KUKA KRL program: ps_604ac_c1.src, ps_604ac_c1.dat

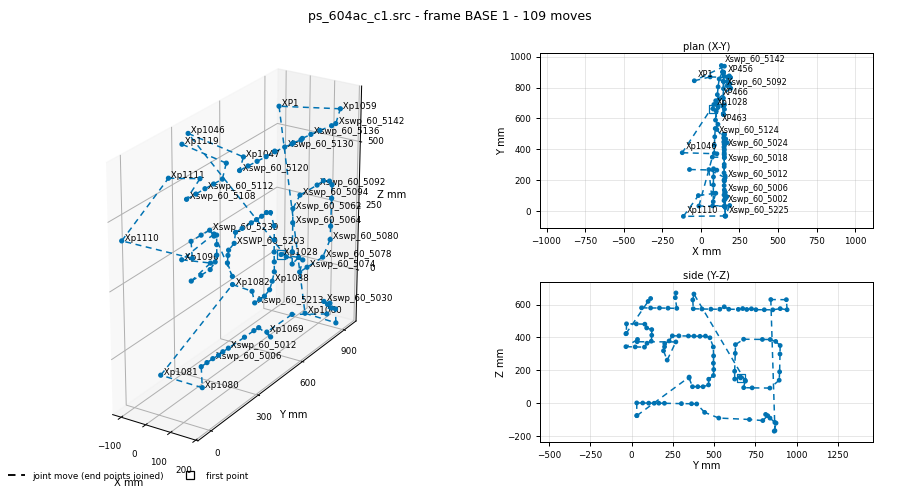
[picture p0: tool path of ps_604ac_c1.src in frame BASE 1, 109 of 111 moves have a stored position in this frame; points joined in program order, loops and branches not executed]
--- ps_604ac_c1.src ---
&ACCESS RVO1
&REL 76
&COMMENT Resp C1 Actros
DEF ps_604ac_c1( )
EXT e_Fraes1 ( )
EXT f_Fraes1 ( )
  ;FOLD INI;%{PE}%V2.2.2,%MKUKATPBASIS,%CINIT,%VCOMMON,%P
  ;FOLD BAS INI;%{PE}%V2.2.2,%MKUKATPBASIS,%CINIT,%VINIT,%P
  INTERRUPT DECL 3 WHEN $STOPMESS==TRUE DO IR_STOPM ( )
  INTERRUPT ON 3
  BAS (#INITMOV,0 )
  ;ENDFOLD
  ;FOLD A20 INI;%{E}%V2.2.2,%MKUKATPA20,%CINIT,%VINIT,%P
  IF ARC20==TRUE THEN
    A20 (ARC_INI)
    INTERRUPT DECL 6 WHEN $CYCFLAG[3]==FALSE DO A20(TECH_STOP2)
  ENDIF
  ;ENDFOLD
  ;FOLD A10 INI;%{E}%V2.2.2,%MKUKATPARC,%CINIT,%VINIT,%P
  IF A10_OPTION==#ACTIVE THEN
    INTERRUPT DECL 4 WHEN $CYCFLAG[2]==FALSE DO A10 (#APPL_ERROR)
    INTERRUPT DECL 7 WHEN A_ARC_SWI==#ACTIVE DO A10 (#ARC_SEAM)
    INTERRUPT DECL 5 WHEN A_FLY_ARC==TRUE DO A10 (#HPU_ARC)
    INTERRUPT  ON 5
    A10_INI ( )
  ENDIF
  ;ENDFOLD
  ;FOLD GRIPPER INI;%{E}%V2.2.2,%MKUKATPGRIPPER,%CINIT,%VINIT,%P
  USER_GRP(0,DUMMY,DUMMY,GDEFAULT)
  ;ENDFOLD
  ;FOLD SPOT INI;%{E}%V.2.2,%MKUKATPSPOT,%CINIT,%VINIT,%P
  USERSPOT(#INIT)
  ;ENDFOLD
  ;FOLD TOUCHSENSE INI;%{E}%V2.2.2,%MKUKATPTS,%CINIT,%VINIT,%P
  IF H70_OPTION THEN
    INTERRUPT DECL 15 WHEN $MEAS_PULSE[TOUCH_I[TOUCH_ACTIVE].IN_NR] DO H70 (6,CD0 )
    INTERRUPT DECL 16 WHEN $ZERO_MOVE DO H70 (7,CD0 )
    INTERRUPT DECL 17 WHEN $TECHPAR_C[FG_TOUCH,8]>0.5 DO H70 (8,CD0)
    H70 (1,CD0 )
  ENDIF
  ;ENDFOLD
  ;FOLD USER INI;%{P}%V2.2.2,%MKUKATPUSER,%CINIT,%VINIT,%P
  ;Make your modifications here
  ;ENDFOLD
  ;ENDFOLD

; Caracterização dos meios de produção: P13.060-R4
; Versão atual: 20/07/2013 12:00  Nome: Solda Respot C1
; Change: Actros

chk_w1_wechs_ok ( )     ; VERIFICAÇÃO DE FERRAMENTA: C1

;FOLD PTP HOME  Vel= 100 % DEFAULT;%{PE}%R 4.1.16,%MKUKATPBASIS,%CMOVE,%VPTP,%P 1:PTP, 2:HOME, 3:, 5:100, 7:DEFAULT
$BWDSTART = FALSE
PDAT_ACT=PDEFAULT
BAS(#PTP_DAT)
FDAT_ACT=FHOME
BAS(#FRAMES)
BAS(#VEL_PTP,100)
$H_POS=XHOME
PTP XHOME
;ENDFOLD

;FOLD OUT 837 'Solic. Lib. Soldar Respot Geo2'  State= TRUE ;%{PE}%R 4.1.16,%MKUKATPBASIS,%COUT,%VOUTX,%P 2:837, 3:'Solic. Lib. Soldar Respot Geo2', 5:TRUE, 6:
$OUT[837]=TRUE
;ENDFOLD
;FOLD WAIT FOR IN 844 'R4 Aguard lib soldar RES accelo/actros'  State= TRUE ;%{PE}%R 4.1.16,%MKUKATPBASIS,%CWAIT_FOR,%VWAIT_FOR,%P 1:0, 2:844, 3:'R4 Aguard lib soldar RES accelo/actros', 5:TRUE, 6:
WAIT FOR $IN[844]==TRUE
;ENDFOLD
;FOLD OUT 837 'Solic. Lib. Soldar Respot Geo2'  State= FALSE ;%{PE}%R 4.1.16,%MKUKATPBASIS,%COUT,%VOUTX,%P 2:837, 3:'Solic. Lib. Soldar Respot Geo2', 5:FALSE, 6:
$OUT[837]=FALSE
;ENDFOLD

;FOLD OUT 851 'Libera AGV'  State= FALSE ;%{PE}%R 4.1.16,%MKUKATPBASIS,%COUT,%VOUTX,%P 2:851, 3:'Libera AGV', 5:FALSE, 6:
$OUT[851]=FALSE
;ENDFOLD


;FOLD PTP p1028 CONT Vel= 65 % P_OLP2 Tool[1]:GUN C1 Base[1]:Actros ;%{PE}%R 4.1.16,%MKUKATPBASIS,%CMOVE,%VPTP,%P 1:PTP, 2:p1028, 3:C_PTP, 5:65, 7:P_OLP2
$BWDSTART = FALSE
PDAT_ACT=PP_OLP2
BAS(#PTP_DAT)
FDAT_ACT=Fp1028
BAS(#FRAMES)
BAS(#VEL_PTP,65)
PTP Xp1028 C_PTP
;ENDFOLD

;FOLD OUT 839 'R4 Soldando'  State= TRUE ;%{PE}%R 4.1.16,%MKUKATPBASIS,%COUT,%VOUTX,%P 2:839, 3:'R4 Soldando', 5:TRUE, 6:
$OUT[839]=TRUE
;ENDFOLD
;FOLD OUT 848 'Area de Solda'  State= FALSE ;%{PE}%R 4.1.16,%MKUKATPBASIS,%COUT,%VOUTX,%P 2:848, 3:'Area de Solda', 5:FALSE, 6:
$OUT[848]=FALSE
;ENDFOLD

;FOLD PTP p1029 CONT Vel= 60 % P_OLP3 Tool[1]:GUN C1 Base[1]:Actros ;%{PE}%R 4.1.16,%MKUKATPBASIS,%CMOVE,%VPTP,%P 1:PTP, 2:p1029, 3:C_PTP, 5:60, 7:P_OLP3
$BWDSTART = FALSE
PDAT_ACT=PP_OLP3
BAS(#PTP_DAT)
FDAT_ACT=Fp1029
BAS(#FRAMES)
BAS(#VEL_PTP,60)
PTP Xp1029 C_PTP
;ENDFOLD

;FOLD ; SWP_60_5070;%{PE}%R2.2,%MKUKATPBASIS,%CCOMMENT,%VNORMAL,%P 2: SWP_60_5070
;ENDFOLD
;FOLD PTP swp_60_5070 PDAT2 SPOT Gun= 1 RETR CLS PgNo1= 45 ACTIVE= 1 Tool[1]:GUN C1 Base[1]:Actros ;%{PE}%R 4.1.12,%MKUKATPSPOT,%CSPOT,%VPTP,%P 1:PTP, 2:swp_60_5070, 3:, 5:100, 7:PDAT2, 10:1, 12:#FIRST, 14:#CLO, 16:45, 18:1, 20:0, 22:0, 24:1, 25:NORMAL
$BWDSTART = FALSE
PDAT_ACT=PPDAT2
BAS(#PTP_DAT)
FDAT_ACT=Fswp_60_5070
BAS(#FRAMES)
BAS(#VEL_PTP,PPDAT2.VEL)
S_ACT.GUN=1
S_ACT.PAIR=SDEFAULT.PAIR
S_ACT.RETR=#CLO
S_ACT.CLO_TM=1
S_ACT.PGNO1=45
S_ACT.PGNO2=SDEFAULT.PGNO2
S_ACT.PRESS1=SDEFAULT.PRESS1
S_ACT.PRESS2=SDEFAULT.PRESS2
S_READY=FALSE
PTP Xswp_60_5070
USERSPOT(#SPOT, S_ACT)
WAIT FOR S_READY
;ENDFOLD

;FOLD ; SWP_60_5068;%{PE}%R2.2,%MKUKATPBASIS,%CCOMMENT,%VNORMAL,%P 2: SWP_60_5068
;ENDFOLD
;FOLD PTP swp_60_5068 PDAT3 SPOT Gun= 1 RETR CLS PgNo1= 46 ACTIVE= 1 Tool[1]:GUN C1 Base[1]:Actros ;%{PE}%R 4.1.12,%MKUKATPSPOT,%CSPOT,%VPTP,%P 1:PTP, 2:swp_60_5068, 3:, 5:100, 7:PDAT3, 10:1, 12:#FIRST, 14:#CLO, 16:46, 18:1, 20:0, 22:0, 24:1, 25:NORMAL
$BWDSTART = FALSE
PDAT_ACT=PPDAT3
BAS(#PTP_DAT)
FDAT_ACT=Fswp_60_5068
BAS(#FRAMES)
BAS(#VEL_PTP,PPDAT3.VEL)
S_ACT.GUN=1
S_ACT.PAIR=SDEFAULT.PAIR
S_ACT.RETR=#CLO
S_ACT.CLO_TM=1
S_ACT.PGNO1=46
S_ACT.PGNO2=SDEFAULT.PGNO2
S_ACT.PRESS1=SDEFAULT.PRESS1
S_ACT.PRESS2=SDEFAULT.PRESS2
S_READY=FALSE
PTP Xswp_60_5068
USERSPOT(#SPOT, S_ACT)
WAIT FOR S_READY
;ENDFOLD

;FOLD ; SWP_60_5064;%{PE}%R2.2,%MKUKATPBASIS,%CCOMMENT,%VNORMAL,%P 2: SWP_60_5064
;ENDFOLD
;FOLD PTP swp_60_5064 PDAT4 SPOT Gun= 1 RETR CLS PgNo1= 47 ACTIVE= 1 Tool[1]:GUN C1 Base[1]:Actros ;%{PE}%R 4.1.12,%MKUKATPSPOT,%CSPOT,%VPTP,%P 1:PTP, 2:swp_60_5064, 3:, 5:100, 7:PDAT4, 10:1, 12:#FIRST, 14:#CLO, 16:47, 18:1, 20:0, 22:0, 24:1, 25:NORMAL
$BWDSTART = FALSE
PDAT_ACT=PPDAT4
BAS(#PTP_DAT)
FDAT_ACT=Fswp_60_5064
BAS(#FRAMES)
BAS(#VEL_PTP,PPDAT4.VEL)
S_ACT.GUN=1
S_ACT.PAIR=SDEFAULT.PAIR
S_ACT.RETR=#CLO
S_ACT.CLO_TM=1
S_ACT.PGNO1=47
S_ACT.PGNO2=SDEFAULT.PGNO2
S_ACT.PRESS1=SDEFAULT.PRESS1
S_ACT.PRESS2=SDEFAULT.PRESS2
S_READY=FALSE
PTP Xswp_60_5064
USERSPOT(#SPOT, S_ACT)
WAIT FOR S_READY
;ENDFOLD

;FOLD ; SWP_60_5062;%{PE}%R2.2,%MKUKATPBASIS,%CCOMMENT,%VNORMAL,%P 2: SWP_60_5062
;ENDFOLD
;FOLD PTP swp_60_5062 PDAT5 SPOT Gun= 1 RETR CLS PgNo1= 48 ACTIVE= 1 Tool[1]:GUN C1 Base[1]:Actros ;%{PE}%R 4.1.12,%MKUKATPSPOT,%CSPOT,%VPTP,%P 1:PTP, 2:swp_60_5062, 3:, 5:100, 7:PDAT5, 10:1, 12:#FIRST, 14:#CLO, 16:48, 18:1, 20:0, 22:0, 24:1, 25:NORMAL
$BWDSTART = FALSE
PDAT_ACT=PPDAT5
BAS(#PTP_DAT)
FDAT_ACT=Fswp_60_5062
BAS(#FRAMES)
BAS(#VEL_PTP,PPDAT5.VEL)
S_ACT.GUN=1
S_ACT.PAIR=SDEFAULT.PAIR
S_ACT.RETR=#CLO
S_ACT.CLO_TM=1
S_ACT.PGNO1=48
S_ACT.PGNO2=SDEFAULT.PGNO2
S_ACT.PRESS1=SDEFAULT.PRESS1
S_ACT.PRESS2=SDEFAULT.PRESS2
S_READY=FALSE
PTP Xswp_60_5062
USERSPOT(#SPOT, S_ACT)
WAIT FOR S_READY
;ENDFOLD

;FOLD ; SWP_60_5094;%{PE}%R2.2,%MKUKATPBASIS,%CCOMMENT,%VNORMAL,%P 2: SWP_60_5094
;ENDFOLD
;FOLD PTP swp_60_5094 PDAT6 SPOT Gun= 1 RETR CLS PgNo1= 49 ACTIVE= 1 Tool[1]:GUN C1 Base[1]:Actros ;%{PE}%R 4.1.12,%MKUKATPSPOT,%CSPOT,%VPTP,%P 1:PTP, 2:swp_60_5094, 3:, 5:100, 7:PDAT6, 10:1, 12:#FIRST, 14:#CLO, 16:49, 18:1, 20:0, 22:0, 24:1, 25:NORMAL
$BWDSTART = FALSE
PDAT_ACT=PPDAT6
BAS(#PTP_DAT)
FDAT_ACT=Fswp_60_5094
BAS(#FRAMES)
BAS(#VEL_PTP,PPDAT6.VEL)
S_ACT.GUN=1
S_ACT.PAIR=SDEFAULT.PAIR
S_ACT.RETR=#CLO
S_ACT.CLO_TM=1
S_ACT.PGNO1=49
S_ACT.PGNO2=SDEFAULT.PGNO2
S_ACT.PRESS1=SDEFAULT.PRESS1
S_ACT.PRESS2=SDEFAULT.PRESS2
S_READY=FALSE
PTP Xswp_60_5094
USERSPOT(#SPOT, S_ACT)
WAIT FOR S_READY
;ENDFOLD

;FOLD ; SWP_60_5092;%{PE}%R2.2,%MKUKATPBASIS,%CCOMMENT,%VNORMAL,%P 2: SWP_60_5092
;ENDFOLD
;FOLD PTP swp_60_5092 PDAT7 SPOT Gun= 1 RETR CLS PgNo1= 50 ACTIVE= 1 Tool[1]:GUN C1 Base[1]:Actros ;%{PE}%R 4.1.12,%MKUKATPSPOT,%CSPOT,%VPTP,%P 1:PTP, 2:swp_60_5092, 3:, 5:100, 7:PDAT7, 10:1, 12:#FIRST, 14:#CLO, 16:50, 18:1, 20:0, 22:0, 24:1, 25:NORMAL
$BWDSTART = FALSE
PDAT_ACT=PPDAT7
BAS(#PTP_DAT)
FDAT_ACT=Fswp_60_5092
BAS(#FRAMES)
BAS(#VEL_PTP,PPDAT7.VEL)
S_ACT.GUN=1
S_ACT.PAIR=SDEFAULT.PAIR
S_ACT.RETR=#CLO
S_ACT.CLO_TM=1
S_ACT.PGNO1=50
S_ACT.PGNO2=SDEFAULT.PGNO2
S_ACT.PRESS1=SDEFAULT.PRESS1
S_ACT.PRESS2=SDEFAULT.PRESS2
S_READY=FALSE
PTP Xswp_60_5092
USERSPOT(#SPOT, S_ACT)
WAIT FOR S_READY
;ENDFOLD

;FOLD ; SWP_60_5090;%{PE}%R2.2,%MKUKATPBASIS,%CCOMMENT,%VNORMAL,%P 2: SWP_60_5090
;ENDFOLD
;FOLD PTP swp_60_5090 PDAT8 SPOT Gun= 1 RETR CLS PgNo1= 51 ACTIVE= 1 Tool[1]:GUN C1 Base[1]:Actros ;%{PE}%R 4.1.12,%MKUKATPSPOT,%CSPOT,%VPTP,%P 1:PTP, 2:swp_60_5090, 3:, 5:100, 7:PDAT8, 10:1, 12:#FIRST, 14:#CLO, 16:51, 18:1, 20:0, 22:0, 24:1, 25:NORMAL
$BWDSTART = FALSE
PDAT_ACT=PPDAT8
BAS(#PTP_DAT)
FDAT_ACT=Fswp_60_5090
BAS(#FRAMES)
BAS(#VEL_PTP,PPDAT8.VEL)
S_ACT.GUN=1
S_ACT.PAIR=SDEFAULT.PAIR
S_ACT.RETR=#CLO
S_ACT.CLO_TM=1
S_ACT.PGNO1=51
S_ACT.PGNO2=SDEFAULT.PGNO2
S_ACT.PRESS1=SDEFAULT.PRESS1
S_ACT.PRESS2=SDEFAULT.PRESS2
S_READY=FALSE
PTP Xswp_60_5090
USERSPOT(#SPOT, S_ACT)
WAIT FOR S_READY
;ENDFOLD

;FOLD PTP P456 CONT Vel= 50 % PDAT66 Tool[1]:GUN C1 Base[1]:Actros ;%{PE}%R 4.1.16,%MKUKATPBASIS,%CMOVE,%VPTP,%P 1:PTP, 2:P456, 3:C_PTP, 5:50, 7:PDAT66
$BWDSTART = FALSE
PDAT_ACT=PPDAT66
BAS(#PTP_DAT)
FDAT_ACT=FP456
BAS(#FRAMES)
BAS(#VEL_PTP,50)
PTP XP456 C_PTP
;ENDFOLD

;FOLD ; SWP_60_5088;%{PE}%R2.2,%MKUKATPBASIS,%CCOMMENT,%VNORMAL,%P 2: SWP_60_5088
;ENDFOLD
;FOLD PTP swp_60_5088 PDAT9 SPOT Gun= 1 RETR CLS PgNo1= 52 ACTIVE= 1 Tool[1]:GUN C1 Base[1]:Actros ;%{PE}%R 4.1.12,%MKUKATPSPOT,%CSPOT,%VPTP,%P 1:PTP, 2:swp_60_5088, 3:, 5:100, 7:PDAT9, 10:1, 12:#FIRST, 14:#CLO, 16:52, 18:1, 20:0, 22:0, 24:1, 25:NORMAL
$BWDSTART = FALSE
PDAT_ACT=PPDAT9
BAS(#PTP_DAT)
FDAT_ACT=Fswp_60_5088
BAS(#FRAMES)
BAS(#VEL_PTP,PPDAT9.VEL)
S_ACT.GUN=1
S_ACT.PAIR=SDEFAULT.PAIR
S_ACT.RETR=#CLO
S_ACT.CLO_TM=1
S_ACT.PGNO1=52
S_ACT.PGNO2=SDEFAULT.PGNO2
S_ACT.PRESS1=SDEFAULT.PRESS1
S_ACT.PRESS2=SDEFAULT.PRESS2
S_READY=FALSE
PTP Xswp_60_5088
USERSPOT(#SPOT, S_ACT)
WAIT FOR S_READY
;ENDFOLD

;FOLD ; SWP_60_5086;%{PE}%R2.2,%MKUKATPBASIS,%CCOMMENT,%VNORMAL,%P 2: SWP_60_5086
;ENDFOLD
;FOLD PTP swp_60_5086 PDAT10 SPOT Gun= 1 RETR CLS PgNo1= 53 ACTIVE= 1 Tool[1]:GUN C1 Base[1]:Actros ;%{PE}%R 4.1.12,%MKUKATPSPOT,%CSPOT,%VPTP,%P 1:PTP, 2:swp_60_5086, 3:, 5:100, 7:PDAT10, 10:1, 12:#FIRST, 14:#CLO, 16:53, 18:1, 20:0, 22:0, 24:1, 25:NORMAL
$BWDSTART = FALSE
PDAT_ACT=PPDAT10
BAS(#PTP_DAT)
FDAT_ACT=Fswp_60_5086
BAS(#FRAMES)
BAS(#VEL_PTP,PPDAT10.VEL)
S_ACT.GUN=1
S_ACT.PAIR=SDEFAULT.PAIR
S_ACT.RETR=#CLO
S_ACT.CLO_TM=1
S_ACT.PGNO1=53
S_ACT.PGNO2=SDEFAULT.PGNO2
S_ACT.PRESS1=SDEFAULT.PRESS1
S_ACT.PRESS2=SDEFAULT.PRESS2
S_READY=FALSE
PTP Xswp_60_5086
USERSPOT(#SPOT, S_ACT)
WAIT FOR S_READY
;ENDFOLD

;FOLD ; SWP_60_5082;%{PE}%R2.2,%MKUKATPBASIS,%CCOMMENT,%VNORMAL,%P 2: SWP_60_5082
;ENDFOLD
;FOLD PTP swp_60_5082 PDAT11 SPOT Gun= 1 RETR CLS PgNo1= 54 ACTIVE= 1 Tool[1]:GUN C1 Base[1]:Actros ;%{PE}%R 4.1.12,%MKUKATPSPOT,%CSPOT,%VPTP,%P 1:PTP, 2:swp_60_5082, 3:, 5:100, 7:PDAT11, 10:1, 12:#FIRST, 14:#CLO, 16:54, 18:1, 20:0, 22:0, 24:1, 25:NORMAL
$BWDSTART = FALSE
PDAT_ACT=PPDAT11
BAS(#PTP_DAT)
FDAT_ACT=Fswp_60_5082
BAS(#FRAMES)
BAS(#VEL_PTP,PPDAT11.VEL)
S_ACT.GUN=1
S_ACT.PAIR=SDEFAULT.PAIR
S_ACT.RETR=#CLO
S_ACT.CLO_TM=1
S_ACT.PGNO1=54
S_ACT.PGNO2=SDEFAULT.PGNO2
S_ACT.PRESS1=SDEFAULT.PRESS1
S_ACT.PRESS2=SDEFAULT.PRESS2
S_READY=FALSE
PTP Xswp_60_5082
USERSPOT(#SPOT, S_ACT)
WAIT FOR S_READY
;ENDFOLD

;FOLD ; SWP_60_5080;%{PE}%R2.2,%MKUKATPBASIS,%CCOMMENT,%VNORMAL,%P 2: SWP_60_5080
;ENDFOLD
;FOLD PTP swp_60_5080 PDAT12 SPOT Gun= 1 RETR CLS PgNo1= 55 ACTIVE= 1 Tool[1]:GUN C1 Base[1]:Actros ;%{PE}%R 4.1.12,%MKUKATPSPOT,%CSPOT,%VPTP,%P 1:PTP, 2:swp_60_5080, 3:, 5:100, 7:PDAT12, 10:1, 12:#FIRST, 14:#CLO, 16:55, 18:1, 20:0, 22:0, 24:1, 25:NORMAL
$BWDSTART = FALSE
PDAT_ACT=PPDAT12
BAS(#PTP_DAT)
FDAT_ACT=Fswp_60_5080
BAS(#FRAMES)
BAS(#VEL_PTP,PPDAT12.VEL)
S_ACT.GUN=1
S_ACT.PAIR=SDEFAULT.PAIR
S_ACT.RETR=#CLO
S_ACT.CLO_TM=1
S_ACT.PGNO1=55
S_ACT.PGNO2=SDEFAULT.PGNO2
S_ACT.PRESS1=SDEFAULT.PRESS1
S_ACT.PRESS2=SDEFAULT.PRESS2
S_READY=FALSE
PTP Xswp_60_5080
USERSPOT(#SPOT, S_ACT)
WAIT FOR S_READY
;ENDFOLD

;FOLD ; SWP_60_5078;%{PE}%R2.2,%MKUKATPBASIS,%CCOMMENT,%VNORMAL,%P 2: SWP_60_5078
;ENDFOLD
;FOLD PTP swp_60_5078 PDAT13 SPOT Gun= 1 RETR CLS PgNo1= 56 ACTIVE= 1 Tool[1]:GUN C1 Base[1]:Actros ;%{PE}%R 4.1.12,%MKUKATPSPOT,%CSPOT,%VPTP,%P 1:PTP, 2:swp_60_5078, 3:, 5:100, 7:PDAT13, 10:1, 12:#FIRST, 14:#CLO, 16:56, 18:1, 20:0, 22:0, 24:1, 25:NORMAL
$BWDSTART = FALSE
PDAT_ACT=PPDAT13
BAS(#PTP_DAT)
FDAT_ACT=Fswp_60_5078
BAS(#FRAMES)
BAS(#VEL_PTP,PPDAT13.VEL)
S_ACT.GUN=1
S_ACT.PAIR=SDEFAULT.PAIR
S_ACT.RETR=#CLO
S_ACT.CLO_TM=1
S_ACT.PGNO1=56
S_ACT.PGNO2=SDEFAULT.PGNO2
S_ACT.PRESS1=SDEFAULT.PRESS1
S_ACT.PRESS2=SDEFAULT.PRESS2
S_READY=FALSE
PTP Xswp_60_5078
USERSPOT(#SPOT, S_ACT)
WAIT FOR S_READY
;ENDFOLD

;FOLD ; SWP_60_5074;%{PE}%R2.2,%MKUKATPBASIS,%CCOMMENT,%VNORMAL,%P 2: SWP_60_5074
;ENDFOLD
;FOLD PTP swp_60_5074 PDAT14 SPOT Gun= 1 RETR CLS PgNo1= 57 ACTIVE= 1 Tool[1]:GUN C1 Base[1]:Actros ;%{PE}%R 4.1.12,%MKUKATPSPOT,%CSPOT,%VPTP,%P 1:PTP, 2:swp_60_5074, 3:, 5:100, 7:PDAT14, 10:1, 12:#FIRST, 14:#CLO, 16:57, 18:1, 20:0, 22:0, 24:1, 25:NORMAL
$BWDSTART = FALSE
PDAT_ACT=PPDAT14
BAS(#PTP_DAT)
FDAT_ACT=Fswp_60_5074
BAS(#FRAMES)
BAS(#VEL_PTP,PPDAT14.VEL)
S_ACT.GUN=1
S_ACT.PAIR=SDEFAULT.PAIR
S_ACT.RETR=#CLO
S_ACT.CLO_TM=1
S_ACT.PGNO1=57
S_ACT.PGNO2=SDEFAULT.PGNO2
S_ACT.PRESS1=SDEFAULT.PRESS1
S_ACT.PRESS2=SDEFAULT.PRESS2
S_READY=FALSE
PTP Xswp_60_5074
USERSPOT(#SPOT, S_ACT)
WAIT FOR S_READY
;ENDFOLD

;FOLD ; SWP_60_5072;%{PE}%R2.2,%MKUKATPBASIS,%CCOMMENT,%VNORMAL,%P 2: SWP_60_5072
;ENDFOLD
;FOLD PTP swp_60_5072 PDAT15 SPOT Gun= 1 RETR CLS PgNo1= 58 ACTIVE= 1 Tool[1]:GUN C1 Base[1]:Actros ;%{PE}%R 4.1.12,%MKUKATPSPOT,%CSPOT,%VPTP,%P 1:PTP, 2:swp_60_5072, 3:, 5:100, 7:PDAT15, 10:1, 12:#FIRST, 14:#CLO, 16:58, 18:1, 20:0, 22:0, 24:1, 25:NORMAL
$BWDSTART = FALSE
PDAT_ACT=PPDAT15
BAS(#PTP_DAT)
FDAT_ACT=Fswp_60_5072
BAS(#FRAMES)
BAS(#VEL_PTP,PPDAT15.VEL)
S_ACT.GUN=1
S_ACT.PAIR=SDEFAULT.PAIR
S_ACT.RETR=#CLO
S_ACT.CLO_TM=1
S_ACT.PGNO1=58
S_ACT.PGNO2=SDEFAULT.PGNO2
S_ACT.PRESS1=SDEFAULT.PRESS1
S_ACT.PRESS2=SDEFAULT.PRESS2
S_READY=FALSE
PTP Xswp_60_5072
USERSPOT(#SPOT, S_ACT)
WAIT FOR S_READY
;ENDFOLD

;FOLD PTP p1044 CONT Vel= 60 % P_OLP18 Tool[1]:GUN C1 Base[1]:Actros ;%{PE}%R 4.1.16,%MKUKATPBASIS,%CMOVE,%VPTP,%P 1:PTP, 2:p1044, 3:C_PTP, 5:60, 7:P_OLP18
$BWDSTART = FALSE
PDAT_ACT=PP_OLP18
BAS(#PTP_DAT)
FDAT_ACT=Fp1044
BAS(#FRAMES)
BAS(#VEL_PTP,60)
PTP Xp1044 C_PTP
;ENDFOLD
;FOLD PTP p1045 CONT Vel= 60 % P_OLP19 Tool[1]:GUN C1 Base[1]:Actros ;%{PE}%R 4.1.16,%MKUKATPBASIS,%CMOVE,%VPTP,%P 1:PTP, 2:p1045, 3:C_PTP, 5:60, 7:P_OLP19
$BWDSTART = FALSE
PDAT_ACT=PP_OLP19
BAS(#PTP_DAT)
FDAT_ACT=Fp1045
BAS(#FRAMES)
BAS(#VEL_PTP,60)
PTP Xp1045 C_PTP
;ENDFOLD

;FOLD ; start interlock r3;%{PE}%R 4.1.16,%MKUKATPBASIS,%CCOMMENT,%VNORMAL,%P 2:start interlock r3
;ENDFOLD
;FOLD Kollision.Ueberwachung_3_Ein ;%{PE}%MKUKATPUSER
COLLSTOP( 3, 1 ) ;INTERRUPTUEBERWACHT
;ENDFOLD

;FOLD PTP p1046 CONT Vel= 60 % P_OLP20 Tool[1]:GUN C1 Base[1]:Actros ;%{PE}%R 4.1.16,%MKUKATPBASIS,%CMOVE,%VPTP,%P 1:PTP, 2:p1046, 3:C_PTP, 5:60, 7:P_OLP20
$BWDSTART = FALSE
PDAT_ACT=PP_OLP20
BAS(#PTP_DAT)
FDAT_ACT=Fp1046
BAS(#FRAMES)
BAS(#VEL_PTP,60)
PTP Xp1046 C_PTP
;ENDFOLD
;FOLD PTP p1047 CONT Vel= 60 % P_OLP21 Tool[1]:GUN C1 Base[1]:Actros ;%{PE}%R 4.1.16,%MKUKATPBASIS,%CMOVE,%VPTP,%P 1:PTP, 2:p1047, 3:C_PTP, 5:60, 7:P_OLP21
$BWDSTART = FALSE
PDAT_ACT=PP_OLP21
BAS(#PTP_DAT)
FDAT_ACT=Fp1047
BAS(#FRAMES)
BAS(#VEL_PTP,60)
PTP Xp1047 C_PTP
;ENDFOLD

;FOLD ;  SWP_60_5120;%{PE}%R 4.1.16,%MKUKATPBASIS,%CCOMMENT,%VNORMAL,%P 2: SWP_60_5120
;ENDFOLD
;FOLD PTP swp_60_5120 PDAT16 SPOT Gun= 1 RETR CLS PgNo1= 59 ACTIVE= 1 Tool[1]:GUN C1 Base[1]:Actros ;%{PE}%R 4.1.12,%MKUKATPSPOT,%CSPOT,%VPTP,%P 1:PTP, 2:swp_60_5120, 3:, 5:100, 7:PDAT16, 10:1, 12:#FIRST, 14:#CLO, 16:59, 18:1, 20:0, 22:0, 24:1, 25:NORMAL
$BWDSTART = FALSE
PDAT_ACT=PPDAT16
BAS(#PTP_DAT)
FDAT_ACT=Fswp_60_5120
BAS(#FRAMES)
BAS(#VEL_PTP,PPDAT16.VEL)
S_ACT.GUN=1
S_ACT.PAIR=SDEFAULT.PAIR
S_ACT.RETR=#CLO
S_ACT.CLO_TM=1
S_ACT.PGNO1=59
S_ACT.PGNO2=SDEFAULT.PGNO2
S_ACT.PRESS1=SDEFAULT.PRESS1
S_ACT.PRESS2=SDEFAULT.PRESS2
S_READY=FALSE
PTP Xswp_60_5120
USERSPOT(#SPOT, S_ACT)
WAIT FOR S_READY
;ENDFOLD

;FOLD ; SWP_60_5122;%{PE}%R2.2,%MKUKATPBASIS,%CCOMMENT,%VNORMAL,%P 2: SWP_60_5122
;ENDFOLD
;FOLD PTP swp_60_5122 PDAT17 SPOT Gun= 1 RETR CLS PgNo1= 60 ACTIVE= 1 Tool[1]:GUN C1 Base[1]:Actros ;%{PE}%R 4.1.12,%MKUKATPSPOT,%CSPOT,%VPTP,%P 1:PTP, 2:swp_60_5122, 3:, 5:100, 7:PDAT17, 10:1, 12:#FIRST, 14:#CLO, 16:60, 18:1, 20:0, 22:0, 24:1, 25:NORMAL
$BWDSTART = FALSE
PDAT_ACT=PPDAT17
BAS(#PTP_DAT)
FDAT_ACT=Fswp_60_5122
BAS(#FRAMES)
BAS(#VEL_PTP,PPDAT17.VEL)
S_ACT.GUN=1
S_ACT.PAIR=SDEFAULT.PAIR
S_ACT.RETR=#CLO
S_ACT.CLO_TM=1
S_ACT.PGNO1=60
S_ACT.PGNO2=SDEFAULT.PGNO2
S_ACT.PRESS1=SDEFAULT.PRESS1
S_ACT.PRESS2=SDEFAULT.PRESS2
S_READY=FALSE
PTP Xswp_60_5122
USERSPOT(#SPOT, S_ACT)
WAIT FOR S_READY
;ENDFOLD

;FOLD ; SWP_60_5124;%{PE}%R2.2,%MKUKATPBASIS,%CCOMMENT,%VNORMAL,%P 2: SWP_60_5124
;ENDFOLD
;FOLD PTP swp_60_5124 PDAT18 SPOT Gun= 1 RETR CLS PgNo1= 61 ACTIVE= 1 Tool[1]:GUN C1 Base[1]:Actros ;%{PE}%R 4.1.12,%MKUKATPSPOT,%CSPOT,%VPTP,%P 1:PTP, 2:swp_60_5124, 3:, 5:100, 7:PDAT18, 10:1, 12:#FIRST, 14:#CLO, 16:61, 18:1, 20:0, 22:0, 24:1, 25:NORMAL
$BWDSTART = FALSE
PDAT_ACT=PPDAT18
BAS(#PTP_DAT)
FDAT_ACT=Fswp_60_5124
BAS(#FRAMES)
BAS(#VEL_PTP,PPDAT18.VEL)
S_ACT.GUN=1
S_ACT.PAIR=SDEFAULT.PAIR
S_ACT.RETR=#CLO
S_ACT.CLO_TM=1
S_ACT.PGNO1=61
S_ACT.PGNO2=SDEFAULT.PGNO2
S_ACT.PRESS1=SDEFAULT.PRESS1
S_ACT.PRESS2=SDEFAULT.PRESS2
S_READY=FALSE
PTP Xswp_60_5124
USERSPOT(#SPOT, S_ACT)
WAIT FOR S_READY
;ENDFOLD

;FOLD ; SWP_60_5126;%{PE}%R2.2,%MKUKATPBASIS,%CCOMMENT,%VNORMAL,%P 2: SWP_60_5126
;ENDFOLD
;FOLD PTP swp_60_5126 PDAT19 SPOT Gun= 1 RETR CLS PgNo1= 62 ACTIVE= 1 Tool[1]:GUN C1 Base[1]:Actros ;%{PE}%R 4.1.12,%MKUKATPSPOT,%CSPOT,%VPTP,%P 1:PTP, 2:swp_60_5126, 3:, 5:100, 7:PDAT19, 10:1, 12:#FIRST, 14:#CLO, 16:62, 18:1, 20:0, 22:0, 24:1, 25:NORMAL
$BWDSTART = FALSE
PDAT_ACT=PPDAT19
BAS(#PTP_DAT)
FDAT_ACT=Fswp_60_5126
BAS(#FRAMES)
BAS(#VEL_PTP,PPDAT19.VEL)
S_ACT.GUN=1
S_ACT.PAIR=SDEFAULT.PAIR
S_ACT.RETR=#CLO
S_ACT.CLO_TM=1
S_ACT.PGNO1=62
S_ACT.PGNO2=SDEFAULT.PGNO2
S_ACT.PRESS1=SDEFAULT.PRESS1
S_ACT.PRESS2=SDEFAULT.PRESS2
S_READY=FALSE
PTP Xswp_60_5126
USERSPOT(#SPOT, S_ACT)
WAIT FOR S_READY
;ENDFOLD

;FOLD PTP P463 CONT Vel= 70 % PDAT72 Tool[1]:GUN C1 Base[1]:Actros ;%{PE}%R 4.1.16,%MKUKATPBASIS,%CMOVE,%VPTP,%P 1:PTP, 2:P463, 3:C_PTP, 5:70, 7:PDAT72
$BWDSTART = FALSE
PDAT_ACT=PPDAT72
BAS(#PTP_DAT)
FDAT_ACT=FP463
BAS(#FRAMES)
BAS(#VEL_PTP,70)
PTP XP463 C_PTP
;ENDFOLD

;FOLD ; SWP_60_5128;%{PE}%R2.2,%MKUKATPBASIS,%CCOMMENT,%VNORMAL,%P 2: SWP_60_5128
;ENDFOLD
;FOLD PTP swp_60_5128 PDAT20 SPOT Gun= 1 RETR CLS PgNo1= 63 ACTIVE= 1 Tool[1]:GUN C1 Base[1]:Actros ;%{PE}%R 4.1.12,%MKUKATPSPOT,%CSPOT,%VPTP,%P 1:PTP, 2:swp_60_5128, 3:, 5:100, 7:PDAT20, 10:1, 12:#FIRST, 14:#CLO, 16:63, 18:1, 20:0, 22:0, 24:1, 25:NORMAL
$BWDSTART = FALSE
PDAT_ACT=PPDAT20
BAS(#PTP_DAT)
FDAT_ACT=Fswp_60_5128
BAS(#FRAMES)
BAS(#VEL_PTP,PPDAT20.VEL)
S_ACT.GUN=1
S_ACT.PAIR=SDEFAULT.PAIR
S_ACT.RETR=#CLO
S_ACT.CLO_TM=1
S_ACT.PGNO1=63
S_ACT.PGNO2=SDEFAULT.PGNO2
S_ACT.PRESS1=SDEFAULT.PRESS1
S_ACT.PRESS2=SDEFAULT.PRESS2
S_READY=FALSE
PTP Xswp_60_5128
USERSPOT(#SPOT, S_ACT)
WAIT FOR S_READY
;ENDFOLD

;FOLD ; SWP_60_5130;%{PE}%R2.2,%MKUKATPBASIS,%CCOMMENT,%VNORMAL,%P 2: SWP_60_5130
;ENDFOLD
;FOLD PTP swp_60_5130 PDAT21 SPOT Gun= 1 RETR CLS PgNo1= 64 ACTIVE= 1 Tool[1]:GUN C1 Base[1]:Actros ;%{PE}%R 4.1.12,%MKUKATPSPOT,%CSPOT,%VPTP,%P 1:PTP, 2:swp_60_5130, 3:, 5:100, 7:PDAT21, 10:1, 12:#FIRST, 14:#CLO, 16:64, 18:1, 20:0, 22:0, 24:1, 25:NORMAL
$BWDSTART = FALSE
PDAT_ACT=PPDAT21
BAS(#PTP_DAT)
FDAT_ACT=Fswp_60_5130
BAS(#FRAMES)
BAS(#VEL_PTP,PPDAT21.VEL)
S_ACT.GUN=1
S_ACT.PAIR=SDEFAULT.PAIR
S_ACT.RETR=#CLO
S_ACT.CLO_TM=1
S_ACT.PGNO1=64
S_ACT.PGNO2=SDEFAULT.PGNO2
S_ACT.PRESS1=SDEFAULT.PRESS1
S_ACT.PRESS2=SDEFAULT.PRESS2
S_READY=FALSE
PTP Xswp_60_5130
USERSPOT(#SPOT, S_ACT)
WAIT FOR S_READY
;ENDFOLD

;FOLD PTP P465 CONT Vel= 70 % PDAT74 Tool[1]:GUN C1 Base[1]:Actros ;%{PE}%R 4.1.16,%MKUKATPBASIS,%CMOVE,%VPTP,%P 1:PTP, 2:P465, 3:C_PTP, 5:70, 7:PDAT74
$BWDSTART = FALSE
PDAT_ACT=PPDAT74
BAS(#PTP_DAT)
FDAT_ACT=FP465
BAS(#FRAMES)
BAS(#VEL_PTP,70)
PTP XP465 C_PTP
;ENDFOLD

;FOLD ; SWP_60_5132;%{PE}%R2.2,%MKUKATPBASIS,%CCOMMENT,%VNORMAL,%P 2: SWP_60_5132
;ENDFOLD
;FOLD PTP swp_60_5132 PDAT22 SPOT Gun= 1 RETR CLS PgNo1= 65 ACTIVE= 1 Tool[1]:GUN C1 Base[1]:Actros ;%{PE}%R 4.1.12,%MKUKATPSPOT,%CSPOT,%VPTP,%P 1:PTP, 2:swp_60_5132, 3:, 5:100, 7:PDAT22, 10:1, 12:#FIRST, 14:#CLO, 16:65, 18:1, 20:0, 22:0, 24:1, 25:NORMAL
$BWDSTART = FALSE
PDAT_ACT=PPDAT22
BAS(#PTP_DAT)
FDAT_ACT=Fswp_60_5132
BAS(#FRAMES)
BAS(#VEL_PTP,PPDAT22.VEL)
S_ACT.GUN=1
S_ACT.PAIR=SDEFAULT.PAIR
S_ACT.RETR=#CLO
S_ACT.CLO_TM=1
S_ACT.PGNO1=65
S_ACT.PGNO2=SDEFAULT.PGNO2
S_ACT.PRESS1=SDEFAULT.PRESS1
S_ACT.PRESS2=SDEFAULT.PRESS2
S_READY=FALSE
PTP Xswp_60_5132
USERSPOT(#SPOT, S_ACT)
WAIT FOR S_READY
;ENDFOLD

;FOLD PTP P466 CONT Vel= 70 % PDAT75 Tool[1]:GUN C1 Base[1]:Actros ;%{PE}%R 4.1.16,%MKUKATPBASIS,%CMOVE,%VPTP,%P 1:PTP, 2:P466, 3:C_PTP, 5:70, 7:PDAT75
$BWDSTART = FALSE
PDAT_ACT=PPDAT75
BAS(#PTP_DAT)
FDAT_ACT=FP466
BAS(#FRAMES)
BAS(#VEL_PTP,70)
PTP XP466 C_PTP
;ENDFOLD

;FOLD ; SWP_60_5134;%{PE}%R2.2,%MKUKATPBASIS,%CCOMMENT,%VNORMAL,%P 2: SWP_60_5134
;ENDFOLD
;FOLD PTP swp_60_5134 PDAT23 SPOT Gun= 1 RETR CLS PgNo1= 66 ACTIVE= 1 Tool[1]:GUN C1 Base[1]:Actros ;%{PE}%R 4.1.12,%MKUKATPSPOT,%CSPOT,%VPTP,%P 1:PTP, 2:swp_60_5134, 3:, 5:100, 7:PDAT23, 10:1, 12:#FIRST, 14:#CLO, 16:66, 18:1, 20:0, 22:0, 24:1, 25:NORMAL
$BWDSTART = FALSE
PDAT_ACT=PPDAT23
BAS(#PTP_DAT)
FDAT_ACT=Fswp_60_5134
BAS(#FRAMES)
BAS(#VEL_PTP,PPDAT23.VEL)
S_ACT.GUN=1
S_ACT.PAIR=SDEFAULT.PAIR
S_ACT.RETR=#CLO
S_ACT.CLO_TM=1
S_ACT.PGNO1=66
S_ACT.PGNO2=SDEFAULT.PGNO2
S_ACT.PRESS1=SDEFAULT.PRESS1
S_ACT.PRESS2=SDEFAULT.PRESS2
S_READY=FALSE
PTP Xswp_60_5134
USERSPOT(#SPOT, S_ACT)
WAIT FOR S_READY
;ENDFOLD

;FOLD ; end interlock r3;%{PE}%R 4.1.16,%MKUKATPBASIS,%CCOMMENT,%VNORMAL,%P 2:end interlock r3
;ENDFOLD
;FOLD Kollision.Ueberwachung_3_Aus ;%{PE}%MKUKATPUSER
COLLSTOP( 3, 2 )
;ENDFOLD

;FOLD ; SWP_60_5136;%{PE}%R2.2,%MKUKATPBASIS,%CCOMMENT,%VNORMAL,%P 2: SWP_60_5136
;ENDFOLD
;FOLD PTP swp_60_5136 PDAT24 SPOT Gun= 1 RETR CLS PgNo1= 67 ACTIVE= 1 Tool[1]:GUN C1 Base[1]:Actros ;%{PE}%R 4.1.12,%MKUKATPSPOT,%CSPOT,%VPTP,%P 1:PTP, 2:swp_60_5136, 3:, 5:100, 7:PDAT24, 10:1, 12:#FIRST, 14:#CLO, 16:67, 18:1, 20:0, 22:0, 24:1, 25:NORMAL
$BWDSTART = FALSE
PDAT_ACT=PPDAT24
BAS(#PTP_DAT)
FDAT_ACT=Fswp_60_5136
BAS(#FRAMES)
BAS(#VEL_PTP,PPDAT24.VEL)
S_ACT.GUN=1
S_ACT.PAIR=SDEFAULT.PAIR
S_ACT.RETR=#CLO
S_ACT.CLO_TM=1
S_ACT.PGNO1=67
S_ACT.PGNO2=SDEFAULT.PGNO2
S_ACT.PRESS1=SDEFAULT.PRESS1
S_ACT.PRESS2=SDEFAULT.PRESS2
S_READY=FALSE
PTP Xswp_60_5136
USERSPOT(#SPOT, S_ACT)
WAIT FOR S_READY
;ENDFOLD

;FOLD ; SWP_60_5138;%{PE}%R2.2,%MKUKATPBASIS,%CCOMMENT,%VNORMAL,%P 2: SWP_60_5138
;ENDFOLD
;FOLD PTP swp_60_5138 PDAT25 SPOT Gun= 1 RETR CLS PgNo1= 68 ACTIVE= 1 Tool[1]:GUN C1 Base[1]:Actros ;%{PE}%R 4.1.12,%MKUKATPSPOT,%CSPOT,%VPTP,%P 1:PTP, 2:swp_60_5138, 3:, 5:100, 7:PDAT25, 10:1, 12:#FIRST, 14:#CLO, 16:68, 18:1, 20:0, 22:0, 24:1, 25:NORMAL
$BWDSTART = FALSE
PDAT_ACT=PPDAT25
BAS(#PTP_DAT)
FDAT_ACT=Fswp_60_5138
BAS(#FRAMES)
BAS(#VEL_PTP,PPDAT25.VEL)
S_ACT.GUN=1
S_ACT.PAIR=SDEFAULT.PAIR
S_ACT.RETR=#CLO
S_ACT.CLO_TM=1
S_ACT.PGNO1=68
S_ACT.PGNO2=SDEFAULT.PGNO2
S_ACT.PRESS1=SDEFAULT.PRESS1
S_ACT.PRESS2=SDEFAULT.PRESS2
S_READY=FALSE
PTP Xswp_60_5138
USERSPOT(#SPOT, S_ACT)
WAIT FOR S_READY
;ENDFOLD

;FOLD PTP P467 CONT Vel= 70 % PDAT76 Tool[1]:GUN C1 Base[1]:Actros ;%{PE}%R 4.1.16,%MKUKATPBASIS,%CMOVE,%VPTP,%P 1:PTP, 2:P467, 3:C_PTP, 5:70, 7:PDAT76
$BWDSTART = FALSE
PDAT_ACT=PPDAT76
BAS(#PTP_DAT)
FDAT_ACT=FP467
BAS(#FRAMES)
BAS(#VEL_PTP,70)
PTP XP467 C_PTP
;ENDFOLD

;FOLD ; SWP_60_5142;%{PE}%R2.2,%MKUKATPBASIS,%CCOMMENT,%VNORMAL,%P 2: SWP_60_5142
;ENDFOLD
;FOLD PTP swp_60_5142 PDAT26 SPOT Gun= 1 RETR CLS PgNo1= 69 ACTIVE= 1 Tool[1]:GUN C1 Base[1]:Actros ;%{PE}%R 4.1.12,%MKUKATPSPOT,%CSPOT,%VPTP,%P 1:PTP, 2:swp_60_5142, 3:, 5:100, 7:PDAT26, 10:1, 12:#FIRST, 14:#CLO, 16:69, 18:1, 20:0, 22:0, 24:1, 25:NORMAL
$BWDSTART = FALSE
PDAT_ACT=PPDAT26
BAS(#PTP_DAT)
FDAT_ACT=Fswp_60_5142
BAS(#FRAMES)
BAS(#VEL_PTP,PPDAT26.VEL)
S_ACT.GUN=1
S_ACT.PAIR=SDEFAULT.PAIR
S_ACT.RETR=#CLO
S_ACT.CLO_TM=1
S_ACT.PGNO1=69
S_ACT.PGNO2=SDEFAULT.PGNO2
S_ACT.PRESS1=SDEFAULT.PRESS1
S_ACT.PRESS2=SDEFAULT.PRESS2
S_READY=FALSE
PTP Xswp_60_5142
USERSPOT(#SPOT, S_ACT)
WAIT FOR S_READY
;ENDFOLD

;FOLD PTP p1059 CONT Vel= 60 % P_OLP33 Tool[1]:GUN C1 Base[1]:Actros ;%{PE}%R 4.1.16,%MKUKATPBASIS,%CMOVE,%VPTP,%P 1:PTP, 2:p1059, 3:C_PTP, 5:60, 7:P_OLP33
$BWDSTART = FALSE
PDAT_ACT=PP_OLP33
BAS(#PTP_DAT)
FDAT_ACT=Fp1059
BAS(#FRAMES)
BAS(#VEL_PTP,60)
PTP Xp1059 C_PTP
;ENDFOLD
;FOLD PTP P1 CONT Vel= 65 % PDAT1 Tool[1]:GUN C1 Base[1]:Actros ;%{PE}%R 4.1.16,%MKUKATPBASIS,%CMOVE,%VPTP,%P 1:PTP, 2:P1, 3:C_PTP, 5:65, 7:PDAT1
$BWDSTART = FALSE
PDAT_ACT=PPDAT1
BAS(#PTP_DAT)
FDAT_ACT=FP1
BAS(#FRAMES)
BAS(#VEL_PTP,65)
PTP XP1 C_PTP
;ENDFOLD
;FOLD PTP p1060 CONT Vel= 65 % P_OLP34 Tool[1]:GUN C1 Base[1]:Actros ;%{PE}%R 4.1.16,%MKUKATPBASIS,%CMOVE,%VPTP,%P 1:PTP, 2:p1060, 3:C_PTP, 5:65, 7:P_OLP34
$BWDSTART = FALSE
PDAT_ACT=PP_OLP34
BAS(#PTP_DAT)
FDAT_ACT=Fp1060
BAS(#FRAMES)
BAS(#VEL_PTP,65)
PTP Xp1060 C_PTP
;ENDFOLD
;FOLD PTP p1061 CONT Vel= 60 % P_OLP35 Tool[1]:GUN C1 Base[1]:Actros ;%{PE}%R 4.1.16,%MKUKATPBASIS,%CMOVE,%VPTP,%P 1:PTP, 2:p1061, 3:C_PTP, 5:60, 7:P_OLP35
$BWDSTART = FALSE
PDAT_ACT=PP_OLP35
BAS(#PTP_DAT)
FDAT_ACT=Fp1061
BAS(#FRAMES)
BAS(#VEL_PTP,60)
PTP Xp1061 C_PTP
;ENDFOLD
;FOLD PTP P457 CONT Vel= 50 % PDAT67 Tool[1]:GUN C1 Base[1]:Actros ;%{PE}%R 4.1.16,%MKUKATPBASIS,%CMOVE,%VPTP,%P 1:PTP, 2:P457, 3:C_PTP, 5:50, 7:PDAT67
$BWDSTART = FALSE
PDAT_ACT=PPDAT67
BAS(#PTP_DAT)
FDAT_ACT=FP457
BAS(#FRAMES)
BAS(#VEL_PTP,50)
PTP XP457 C_PTP
;ENDFOLD

;FOLD ; SWP_60_5034;%{PE}%R2.2,%MKUKATPBASIS,%CCOMMENT,%VNORMAL,%P 2: SWP_60_5034
;ENDFOLD
;FOLD PTP swp_60_5034 PDAT27 SPOT Gun= 1 RETR CLS PgNo1= 70 ACTIVE= 1 Tool[1]:GUN C1 Base[1]:Actros ;%{PE}%R 4.1.12,%MKUKATPSPOT,%CSPOT,%VPTP,%P 1:PTP, 2:swp_60_5034, 3:, 5:100, 7:PDAT27, 10:1, 12:#FIRST, 14:#CLO, 16:70, 18:1, 20:0, 22:0, 24:1, 25:NORMAL
$BWDSTART = FALSE
PDAT_ACT=PPDAT27
BAS(#PTP_DAT)
FDAT_ACT=Fswp_60_5034
BAS(#FRAMES)
BAS(#VEL_PTP,PPDAT27.VEL)
S_ACT.GUN=1
S_ACT.PAIR=SDEFAULT.PAIR
S_ACT.RETR=#CLO
S_ACT.CLO_TM=1
S_ACT.PGNO1=70
S_ACT.PGNO2=SDEFAULT.PGNO2
S_ACT.PRESS1=SDEFAULT.PRESS1
S_ACT.PRESS2=SDEFAULT.PRESS2
S_READY=FALSE
PTP Xswp_60_5034
USERSPOT(#SPOT, S_ACT)
WAIT FOR S_READY
;ENDFOLD

;FOLD ; SWP_60_5032;%{PE}%R2.2,%MKUKATPBASIS,%CCOMMENT,%VNORMAL,%P 2: SWP_60_5032
;ENDFOLD
;FOLD PTP swp_60_5032 PDAT28 SPOT Gun= 1 RETR CLS PgNo1= 71 ACTIVE= 1 Tool[1]:GUN C1 Base[1]:Actros ;%{PE}%R 4.1.12,%MKUKATPSPOT,%CSPOT,%VPTP,%P 1:PTP, 2:swp_60_5032, 3:, 5:100, 7:PDAT28, 10:1, 12:#FIRST, 14:#CLO, 16:71, 18:1, 20:0, 22:0, 24:1, 25:NORMAL
$BWDSTART = FALSE
PDAT_ACT=PPDAT28
BAS(#PTP_DAT)
FDAT_ACT=Fswp_60_5032
BAS(#FRAMES)
BAS(#VEL_PTP,PPDAT28.VEL)
S_ACT.GUN=1
S_ACT.PAIR=SDEFAULT.PAIR
S_ACT.RETR=#CLO
S_ACT.CLO_TM=1
S_ACT.PGNO1=71
S_ACT.PGNO2=SDEFAULT.PGNO2
S_ACT.PRESS1=SDEFAULT.PRESS1
S_ACT.PRESS2=SDEFAULT.PRESS2
S_READY=FALSE
PTP Xswp_60_5032
USERSPOT(#SPOT, S_ACT)
WAIT FOR S_READY
;ENDFOLD

;FOLD ; SWP_60_5030;%{PE}%R2.2,%MKUKATPBASIS,%CCOMMENT,%VNORMAL,%P 2: SWP_60_5030
;ENDFOLD
;FOLD PTP swp_60_5030 PDAT29 SPOT Gun= 1 RETR CLS PgNo1= 72 ACTIVE= 1 Tool[1]:GUN C1 Base[1]:Actros ;%{PE}%R 4.1.12,%MKUKATPSPOT,%CSPOT,%VPTP,%P 1:PTP, 2:swp_60_5030, 3:, 5:100, 7:PDAT29, 10:1, 12:#FIRST, 14:#CLO, 16:72, 18:1, 20:0, 22:0, 24:1, 25:NORMAL
$BWDSTART = FALSE
PDAT_ACT=PPDAT29
BAS(#PTP_DAT)
FDAT_ACT=Fswp_60_5030
BAS(#FRAMES)
BAS(#VEL_PTP,PPDAT29.VEL)
S_ACT.GUN=1
S_ACT.PAIR=SDEFAULT.PAIR
S_ACT.RETR=#CLO
S_ACT.CLO_TM=1
S_ACT.PGNO1=72
S_ACT.PGNO2=SDEFAULT.PGNO2
S_ACT.PRESS1=SDEFAULT.PRESS1
S_ACT.PRESS2=SDEFAULT.PRESS2
S_READY=FALSE
PTP Xswp_60_5030
USERSPOT(#SPOT, S_ACT)
WAIT FOR S_READY
;ENDFOLD

;FOLD PTP p1066 CONT Vel= 60 % P_OLP40 Tool[1]:GUN C1 Base[1]:Actros ;%{PE}%R 4.1.16,%MKUKATPBASIS,%CMOVE,%VPTP,%P 1:PTP, 2:p1066, 3:C_PTP, 5:60, 7:P_OLP40
$BWDSTART = FALSE
PDAT_ACT=PP_OLP40
BAS(#PTP_DAT)
FDAT_ACT=Fp1066
BAS(#FRAMES)
BAS(#VEL_PTP,60)
PTP Xp1066 C_PTP
;ENDFOLD
;FOLD PTP p1067 CONT Vel= 70 % P_OLP41 Tool[1]:GUN C1 Base[1]:Actros ;%{PE}%R 4.1.16,%MKUKATPBASIS,%CMOVE,%VPTP,%P 1:PTP, 2:p1067, 3:C_PTP, 5:70, 7:P_OLP41
$BWDSTART = FALSE
PDAT_ACT=PP_OLP41
BAS(#PTP_DAT)
FDAT_ACT=Fp1067
BAS(#FRAMES)
BAS(#VEL_PTP,70)
PTP Xp1067 C_PTP
;ENDFOLD

;FOLD ;  START INTERLOCK COM R3;%{PE}%R 4.1.16,%MKUKATPBASIS,%CCOMMENT,%VNORMAL,%P 2: START INTERLOCK COM R3
;ENDFOLD

;FOLD Kollision.Ueberwachung_3_Ein ;%{PE}%MKUKATPUSER
COLLSTOP( 3, 1 ) ;INTERRUPTUEBERWACHT
;ENDFOLD

;FOLD PTP p1068 CONT Vel= 70 % P_OLP42 Tool[1]:GUN C1 Base[1]:Actros ;%{PE}%R 4.1.16,%MKUKATPBASIS,%CMOVE,%VPTP,%P 1:PTP, 2:p1068, 3:C_PTP, 5:70, 7:P_OLP42
$BWDSTART = FALSE
PDAT_ACT=PP_OLP42
BAS(#PTP_DAT)
FDAT_ACT=Fp1068
BAS(#FRAMES)
BAS(#VEL_PTP,70)
PTP Xp1068 C_PTP
;ENDFOLD
;FOLD PTP p1069 CONT Vel= 70 % P_OLP43 Tool[1]:GUN C1 Base[1]:Actros ;%{PE}%R 4.1.16,%MKUKATPBASIS,%CMOVE,%VPTP,%P 1:PTP, 2:p1069, 3:C_PTP, 5:70, 7:P_OLP43
$BWDSTART = FALSE
PDAT_ACT=PP_OLP43
BAS(#PTP_DAT)
FDAT_ACT=Fp1069
BAS(#FRAMES)
BAS(#VEL_PTP,70)
PTP Xp1069 C_PTP
;ENDFOLD
;FOLD PTP p1070 CONT Vel= 60 % P_OLP44 Tool[1]:GUN C1 Base[1]:Actros ;%{PE}%R 4.1.16,%MKUKATPBASIS,%CMOVE,%VPTP,%P 1:PTP, 2:p1070, 3:C_PTP, 5:60, 7:P_OLP44
$BWDSTART = FALSE
PDAT_ACT=PP_OLP44
BAS(#PTP_DAT)
FDAT_ACT=Fp1070
BAS(#FRAMES)
BAS(#VEL_PTP,60)
PTP Xp1070 C_PTP
;ENDFOLD

;FOLD ; SWP_60_5024;%{PE}%R2.2,%MKUKATPBASIS,%CCOMMENT,%VNORMAL,%P 2: SWP_60_5024
;ENDFOLD
;FOLD PTP swp_60_5024 PDAT30 SPOT Gun= 1 RETR CLS PgNo1= 73 ACTIVE= 1 Tool[1]:GUN C1 Base[1]:Actros ;%{PE}%R 4.1.12,%MKUKATPSPOT,%CSPOT,%VPTP,%P 1:PTP, 2:swp_60_5024, 3:, 5:100, 7:PDAT30, 10:1, 12:#FIRST, 14:#CLO, 16:73, 18:1, 20:0, 22:0, 24:1, 25:NORMAL
$BWDSTART = FALSE
PDAT_ACT=PPDAT30
BAS(#PTP_DAT)
FDAT_ACT=Fswp_60_5024
BAS(#FRAMES)
BAS(#VEL_PTP,PPDAT30.VEL)
S_ACT.GUN=1
S_ACT.PAIR=SDEFAULT.PAIR
S_ACT.RETR=#CLO
S_ACT.CLO_TM=1
S_ACT.PGNO1=73
S_ACT.PGNO2=SDEFAULT.PGNO2
S_ACT.PRESS1=SDEFAULT.PRESS1
S_ACT.PRESS2=SDEFAULT.PRESS2
S_READY=FALSE
PTP Xswp_60_5024
USERSPOT(#SPOT, S_ACT)
WAIT FOR S_READY
;ENDFOLD

;FOLD ; SWP_60_5022;%{PE}%R2.2,%MKUKATPBASIS,%CCOMMENT,%VNORMAL,%P 2: SWP_60_5022
;ENDFOLD
;FOLD PTP swp_60_5022 PDAT31 SPOT Gun= 1 RETR CLS PgNo1= 74 ACTIVE= 1 Tool[1]:GUN C1 Base[1]:Actros ;%{PE}%R 4.1.12,%MKUKATPSPOT,%CSPOT,%VPTP,%P 1:PTP, 2:swp_60_5022, 3:, 5:100, 7:PDAT31, 10:1, 12:#FIRST, 14:#CLO, 16:74, 18:1, 20:0, 22:0, 24:1, 25:NORMAL
$BWDSTART = FALSE
PDAT_ACT=PPDAT31
BAS(#PTP_DAT)
FDAT_ACT=Fswp_60_5022
BAS(#FRAMES)
BAS(#VEL_PTP,PPDAT31.VEL)
S_ACT.GUN=1
S_ACT.PAIR=SDEFAULT.PAIR
S_ACT.RETR=#CLO
S_ACT.CLO_TM=1
S_ACT.PGNO1=74
S_ACT.PGNO2=SDEFAULT.PGNO2
S_ACT.PRESS1=SDEFAULT.PRESS1
S_ACT.PRESS2=SDEFAULT.PRESS2
S_READY=FALSE
PTP Xswp_60_5022
USERSPOT(#SPOT, S_ACT)
WAIT FOR S_READY
;ENDFOLD

;FOLD ; liga interlock r3;%{PE}%R 4.1.16,%MKUKATPBASIS,%CCOMMENT,%VNORMAL,%P 2:liga interlock r3
;ENDFOLD
;FOLD Kollision.Ueberwachung_3_Ein ;%{PE}%MKUKATPUSER
COLLSTOP( 3, 1 ) ;INTERRUPTUEBERWACHT
;ENDFOLD

;FOLD ;  SWP_60_5018;%{PE}%R 4.1.16,%MKUKATPBASIS,%CCOMMENT,%VNORMAL,%P 2: SWP_60_5018
;ENDFOLD
;FOLD PTP swp_60_5018 PDAT65 SPOT Gun= 1 RETR CLS PgNo1= 75 ACTIVE= 1 Tool[1]:GUN C1 Base[1]:Actros ;%{PE}%R 4.1.12,%MKUKATPSPOT,%CSPOT,%VPTP,%P 1:PTP, 2:swp_60_5018, 3:, 5:100, 7:PDAT65, 10:1, 12:#FIRST, 14:#CLO, 16:75, 18:1, 20:0, 22:0, 24:1, 25:NORMAL
$BWDSTART = FALSE
PDAT_ACT=PPDAT65
BAS(#PTP_DAT)
FDAT_ACT=Fswp_60_5018
BAS(#FRAMES)
BAS(#VEL_PTP,PPDAT65.VEL)
S_ACT.GUN=1
S_ACT.PAIR=SDEFAULT.PAIR
S_ACT.RETR=#CLO
S_ACT.CLO_TM=1
S_ACT.PGNO1=75
S_ACT.PGNO2=SDEFAULT.PGNO2
S_ACT.PRESS1=SDEFAULT.PRESS1
S_ACT.PRESS2=SDEFAULT.PRESS2
S_READY=FALSE
PTP Xswp_60_5018
USERSPOT(#SPOT, S_ACT)
WAIT FOR S_READY
;ENDFOLD

;FOLD ; SWP_60_5012;%{PE}%R2.2,%MKUKATPBASIS,%CCOMMENT,%VNORMAL,%P 2: SWP_60_5012
;ENDFOLD
;FOLD PTP swp_60_5012 PDAT33 SPOT Gun= 1 RETR CLS PgNo1= 76 ACTIVE= 1 Tool[1]:GUN C1 Base[1]:Actros ;%{PE}%R 4.1.12,%MKUKATPSPOT,%CSPOT,%VPTP,%P 1:PTP, 2:swp_60_5012, 3:, 5:100, 7:PDAT33, 10:1, 12:#FIRST, 14:#CLO, 16:76, 18:1, 20:0, 22:0, 24:1, 25:NORMAL
$BWDSTART = FALSE
PDAT_ACT=PPDAT33
BAS(#PTP_DAT)
FDAT_ACT=Fswp_60_5012
BAS(#FRAMES)
BAS(#VEL_PTP,PPDAT33.VEL)
S_ACT.GUN=1
S_ACT.PAIR=SDEFAULT.PAIR
S_ACT.RETR=#CLO
S_ACT.CLO_TM=1
S_ACT.PGNO1=76
S_ACT.PGNO2=SDEFAULT.PGNO2
S_ACT.PRESS1=SDEFAULT.PRESS1
S_ACT.PRESS2=SDEFAULT.PRESS2
S_READY=FALSE
PTP Xswp_60_5012
USERSPOT(#SPOT, S_ACT)
WAIT FOR S_READY
;ENDFOLD

;FOLD ; SWP_60_5010;%{PE}%R2.2,%MKUKATPBASIS,%CCOMMENT,%VNORMAL,%P 2: SWP_60_5010
;ENDFOLD
;FOLD PTP swp_60_5010 PDAT34 SPOT Gun= 1 RETR CLS PgNo1= 77 ACTIVE= 1 Tool[1]:GUN C1 Base[1]:Actros ;%{PE}%R 4.1.12,%MKUKATPSPOT,%CSPOT,%VPTP,%P 1:PTP, 2:swp_60_5010, 3:, 5:100, 7:PDAT34, 10:1, 12:#FIRST, 14:#CLO, 16:77, 18:1, 20:0, 22:0, 24:1, 25:NORMAL
$BWDSTART = FALSE
PDAT_ACT=PPDAT34
BAS(#PTP_DAT)
FDAT_ACT=Fswp_60_5010
BAS(#FRAMES)
BAS(#VEL_PTP,PPDAT34.VEL)
S_ACT.GUN=1
S_ACT.PAIR=SDEFAULT.PAIR
S_ACT.RETR=#CLO
S_ACT.CLO_TM=1
S_ACT.PGNO1=77
S_ACT.PGNO2=SDEFAULT.PGNO2
S_ACT.PRESS1=SDEFAULT.PRESS1
S_ACT.PRESS2=SDEFAULT.PRESS2
S_READY=FALSE
PTP Xswp_60_5010
USERSPOT(#SPOT, S_ACT)
WAIT FOR S_READY
;ENDFOLD

;FOLD ; SWP_60_5008;%{PE}%R2.2,%MKUKATPBASIS,%CCOMMENT,%VNORMAL,%P 2: SWP_60_5008
;ENDFOLD
;FOLD PTP swp_60_5008 PDAT35 SPOT Gun= 1 RETR CLS PgNo1= 78 ACTIVE= 1 Tool[1]:GUN C1 Base[1]:Actros ;%{PE}%R 4.1.12,%MKUKATPSPOT,%CSPOT,%VPTP,%P 1:PTP, 2:swp_60_5008, 3:, 5:100, 7:PDAT35, 10:1, 12:#FIRST, 14:#CLO, 16:78, 18:1, 20:0, 22:0, 24:1, 25:NORMAL
$BWDSTART = FALSE
PDAT_ACT=PPDAT35
BAS(#PTP_DAT)
FDAT_ACT=Fswp_60_5008
BAS(#FRAMES)
BAS(#VEL_PTP,PPDAT35.VEL)
S_ACT.GUN=1
S_ACT.PAIR=SDEFAULT.PAIR
S_ACT.RETR=#CLO
S_ACT.CLO_TM=1
S_ACT.PGNO1=78
S_ACT.PGNO2=SDEFAULT.PGNO2
S_ACT.PRESS1=SDEFAULT.PRESS1
S_ACT.PRESS2=SDEFAULT.PRESS2
S_READY=FALSE
PTP Xswp_60_5008
USERSPOT(#SPOT, S_ACT)
WAIT FOR S_READY
;ENDFOLD

;FOLD ; SWP_60_5006;%{PE}%R2.2,%MKUKATPBASIS,%CCOMMENT,%VNORMAL,%P 2: SWP_60_5006
;ENDFOLD
;FOLD PTP swp_60_5006 PDAT36 SPOT Gun= 1 RETR CLS PgNo1= 79 ACTIVE= 1 Tool[1]:GUN C1 Base[1]:Actros ;%{PE}%R 4.1.12,%MKUKATPSPOT,%CSPOT,%VPTP,%P 1:PTP, 2:swp_60_5006, 3:, 5:100, 7:PDAT36, 10:1, 12:#FIRST, 14:#CLO, 16:79, 18:1, 20:0, 22:0, 24:1, 25:NORMAL
$BWDSTART = FALSE
PDAT_ACT=PPDAT36
BAS(#PTP_DAT)
FDAT_ACT=Fswp_60_5006
BAS(#FRAMES)
BAS(#VEL_PTP,PPDAT36.VEL)
S_ACT.GUN=1
S_ACT.PAIR=SDEFAULT.PAIR
S_ACT.RETR=#CLO
S_ACT.CLO_TM=1
S_ACT.PGNO1=79
S_ACT.PGNO2=SDEFAULT.PGNO2
S_ACT.PRESS1=SDEFAULT.PRESS1
S_ACT.PRESS2=SDEFAULT.PRESS2
S_READY=FALSE
PTP Xswp_60_5006
USERSPOT(#SPOT, S_ACT)
WAIT FOR S_READY
;ENDFOLD

;FOLD ; SWP_60_5004;%{PE}%R2.2,%MKUKATPBASIS,%CCOMMENT,%VNORMAL,%P 2: SWP_60_5004
;ENDFOLD
;FOLD PTP swp_60_5004 PDAT37 SPOT Gun= 1 RETR CLS PgNo1= 80 ACTIVE= 1 Tool[1]:GUN C1 Base[1]:Actros ;%{PE}%R 4.1.12,%MKUKATPSPOT,%CSPOT,%VPTP,%P 1:PTP, 2:swp_60_5004, 3:, 5:100, 7:PDAT37, 10:1, 12:#FIRST, 14:#CLO, 16:80, 18:1, 20:0, 22:0, 24:1, 25:NORMAL
$BWDSTART = FALSE
PDAT_ACT=PPDAT37
BAS(#PTP_DAT)
FDAT_ACT=Fswp_60_5004
BAS(#FRAMES)
BAS(#VEL_PTP,PPDAT37.VEL)
S_ACT.GUN=1
S_ACT.PAIR=SDEFAULT.PAIR
S_ACT.RETR=#CLO
S_ACT.CLO_TM=1
S_ACT.PGNO1=80
S_ACT.PGNO2=SDEFAULT.PGNO2
S_ACT.PRESS1=SDEFAULT.PRESS1
S_ACT.PRESS2=SDEFAULT.PRESS2
S_READY=FALSE
PTP Xswp_60_5004
USERSPOT(#SPOT, S_ACT)
WAIT FOR S_READY
;ENDFOLD

;FOLD ; SWP_60_5002;%{PE}%R2.2,%MKUKATPBASIS,%CCOMMENT,%VNORMAL,%P 2: SWP_60_5002
;ENDFOLD
;FOLD PTP swp_60_5002 PDAT38 SPOT Gun= 1 RETR CLS PgNo1= 81 ACTIVE= 1 Tool[1]:GUN C1 Base[1]:Actros ;%{PE}%R 4.1.12,%MKUKATPSPOT,%CSPOT,%VPTP,%P 1:PTP, 2:swp_60_5002, 3:, 5:100, 7:PDAT38, 10:1, 12:#FIRST, 14:#CLO, 16:81, 18:1, 20:0, 22:0, 24:1, 25:NORMAL
$BWDSTART = FALSE
PDAT_ACT=PPDAT38
BAS(#PTP_DAT)
FDAT_ACT=Fswp_60_5002
BAS(#FRAMES)
BAS(#VEL_PTP,PPDAT38.VEL)
S_ACT.GUN=1
S_ACT.PAIR=SDEFAULT.PAIR
S_ACT.RETR=#CLO
S_ACT.CLO_TM=1
S_ACT.PGNO1=81
S_ACT.PGNO2=SDEFAULT.PGNO2
S_ACT.PRESS1=SDEFAULT.PRESS1
S_ACT.PRESS2=SDEFAULT.PRESS2
S_READY=FALSE
PTP Xswp_60_5002
USERSPOT(#SPOT, S_ACT)
WAIT FOR S_READY
;ENDFOLD

;FOLD PTP p1080 CONT Vel= 50 % P_OLP54 Tool[1]:GUN C1 Base[1]:Actros ;%{PE}%R 4.1.16,%MKUKATPBASIS,%CMOVE,%VPTP,%P 1:PTP, 2:p1080, 3:C_PTP, 5:50, 7:P_OLP54
$BWDSTART = FALSE
PDAT_ACT=PP_OLP54
BAS(#PTP_DAT)
FDAT_ACT=Fp1080
BAS(#FRAMES)
BAS(#VEL_PTP,50)
PTP Xp1080 C_PTP
;ENDFOLD
;FOLD PTP p1081 CONT Vel= 60 % P_OLP55 Tool[1]:GUN C1 Base[1]:Actros ;%{PE}%R 4.1.16,%MKUKATPBASIS,%CMOVE,%VPTP,%P 1:PTP, 2:p1081, 3:C_PTP, 5:60, 7:P_OLP55
$BWDSTART = FALSE
PDAT_ACT=PP_OLP55
BAS(#PTP_DAT)
FDAT_ACT=Fp1081
BAS(#FRAMES)
BAS(#VEL_PTP,60)
PTP Xp1081 C_PTP
;ENDFOLD
;FOLD PTP p1082 CONT Vel= 60 % P_OLP56 Tool[1]:GUN C1 Base[1]:Actros ;%{PE}%R 4.1.16,%MKUKATPBASIS,%CMOVE,%VPTP,%P 1:PTP, 2:p1082, 3:C_PTP, 5:60, 7:P_OLP56
$BWDSTART = FALSE
PDAT_ACT=PP_OLP56
BAS(#PTP_DAT)
FDAT_ACT=Fp1082
BAS(#FRAMES)
BAS(#VEL_PTP,60)
PTP Xp1082 C_PTP
;ENDFOLD
;FOLD PTP p1083 CONT Vel= 60 % P_OLP57 Tool[1]:GUN C1 Base[1]:Actros ;%{PE}%R 4.1.16,%MKUKATPBASIS,%CMOVE,%VPTP,%P 1:PTP, 2:p1083, 3:C_PTP, 5:60, 7:P_OLP57
$BWDSTART = FALSE
PDAT_ACT=PP_OLP57
BAS(#PTP_DAT)
FDAT_ACT=Fp1083
BAS(#FRAMES)
BAS(#VEL_PTP,60)
PTP Xp1083 C_PTP
;ENDFOLD

;FOLD ; SWP_60_5213;%{PE}%R2.2,%MKUKATPBASIS,%CCOMMENT,%VNORMAL,%P 2: SWP_60_5213
;ENDFOLD
;FOLD PTP swp_60_5213 PDAT39 SPOT Gun= 1 RETR CLS PgNo1= 82 ACTIVE= 1 Tool[1]:GUN C1 Base[1]:Actros ;%{PE}%R 4.1.12,%MKUKATPSPOT,%CSPOT,%VPTP,%P 1:PTP, 2:swp_60_5213, 3:, 5:100, 7:PDAT39, 10:1, 12:#FIRST, 14:#CLO, 16:82, 18:1, 20:0, 22:0, 24:1, 25:NORMAL
$BWDSTART = FALSE
PDAT_ACT=PPDAT39
BAS(#PTP_DAT)
FDAT_ACT=Fswp_60_5213
BAS(#FRAMES)
BAS(#VEL_PTP,PPDAT39.VEL)
S_ACT.GUN=1
S_ACT.PAIR=SDEFAULT.PAIR
S_ACT.RETR=#CLO
S_ACT.CLO_TM=1
S_ACT.PGNO1=82
S_ACT.PGNO2=SDEFAULT.PGNO2
S_ACT.PRESS1=SDEFAULT.PRESS1
S_ACT.PRESS2=SDEFAULT.PRESS2
S_READY=FALSE
PTP Xswp_60_5213
USERSPOT(#SPOT, S_ACT)
WAIT FOR S_READY
;ENDFOLD


;FOLD ; SWP_60_5212;%{PE}%R2.2,%MKUKATPBASIS,%CCOMMENT,%VNORMAL,%P 2: SWP_60_5212
;ENDFOLD
;FOLD PTP swp_60_5212 PDAT40 SPOT Gun= 1 RETR CLS PgNo1= 83 ACTIVE= 1 Tool[1]:GUN C1 Base[1]:Actros ;%{PE}%R 4.1.12,%MKUKATPSPOT,%CSPOT,%VPTP,%P 1:PTP, 2:swp_60_5212, 3:, 5:100, 7:PDAT40, 10:1, 12:#FIRST, 14:#CLO, 16:83, 18:1, 20:0, 22:0, 24:1, 25:NORMAL
$BWDSTART = FALSE
PDAT_ACT=PPDAT40
BAS(#PTP_DAT)
FDAT_ACT=Fswp_60_5212
BAS(#FRAMES)
BAS(#VEL_PTP,PPDAT40.VEL)
S_ACT.GUN=1
S_ACT.PAIR=SDEFAULT.PAIR
S_ACT.RETR=#CLO
S_ACT.CLO_TM=1
S_ACT.PGNO1=83
S_ACT.PGNO2=SDEFAULT.PGNO2
S_ACT.PRESS1=SDEFAULT.PRESS1
S_ACT.PRESS2=SDEFAULT.PRESS2
S_READY=FALSE
PTP Xswp_60_5212
USERSPOT(#SPOT, S_ACT)
WAIT FOR S_READY
;ENDFOLD

;FOLD ; SWP_60_5211;%{PE}%R2.2,%MKUKATPBASIS,%CCOMMENT,%VNORMAL,%P 2: SWP_60_5211
;ENDFOLD
;FOLD PTP swp_60_5211 PDAT41 SPOT Gun= 1 RETR CLS PgNo1= 84 ACTIVE= 1 Tool[1]:GUN C1 Base[1]:Actros ;%{PE}%R 4.1.12,%MKUKATPSPOT,%CSPOT,%VPTP,%P 1:PTP, 2:swp_60_5211, 3:, 5:100, 7:PDAT41, 10:1, 12:#FIRST, 14:#CLO, 16:84, 18:1, 20:0, 22:0, 24:1, 25:NORMAL
$BWDSTART = FALSE
PDAT_ACT=PPDAT41
BAS(#PTP_DAT)
FDAT_ACT=Fswp_60_5211
BAS(#FRAMES)
BAS(#VEL_PTP,PPDAT41.VEL)
S_ACT.GUN=1
S_ACT.PAIR=SDEFAULT.PAIR
S_ACT.RETR=#CLO
S_ACT.CLO_TM=1
S_ACT.PGNO1=84
S_ACT.PGNO2=SDEFAULT.PGNO2
S_ACT.PRESS1=SDEFAULT.PRESS1
S_ACT.PRESS2=SDEFAULT.PRESS2
S_READY=FALSE
PTP Xswp_60_5211
USERSPOT(#SPOT, S_ACT)
WAIT FOR S_READY
;ENDFOLD

;FOLD ; SWP_60_5210;%{PE}%R2.2,%MKUKATPBASIS,%CCOMMENT,%VNORMAL,%P 2: SWP_60_5210
;ENDFOLD
;FOLD PTP swp_60_5210 PDAT42 SPOT Gun= 1 RETR CLS PgNo1= 85 ACTIVE= 1 Tool[1]:GUN C1 Base[1]:Actros ;%{PE}%R 4.1.12,%MKUKATPSPOT,%CSPOT,%VPTP,%P 1:PTP, 2:swp_60_5210, 3:, 5:100, 7:PDAT42, 10:1, 12:#FIRST, 14:#CLO, 16:85, 18:1, 20:0, 22:0, 24:1, 25:NORMAL
$BWDSTART = FALSE
PDAT_ACT=PPDAT42
BAS(#PTP_DAT)
FDAT_ACT=Fswp_60_5210
BAS(#FRAMES)
BAS(#VEL_PTP,PPDAT42.VEL)
S_ACT.GUN=1
S_ACT.PAIR=SDEFAULT.PAIR
S_ACT.RETR=#CLO
S_ACT.CLO_TM=1
S_ACT.PGNO1=85
S_ACT.PGNO2=SDEFAULT.PGNO2
S_ACT.PRESS1=SDEFAULT.PRESS1
S_ACT.PRESS2=SDEFAULT.PRESS2
S_READY=FALSE
PTP Xswp_60_5210
USERSPOT(#SPOT, S_ACT)
WAIT FOR S_READY
;ENDFOLD

;FOLD PTP p1088 CONT Vel= 50 % P_OLP62 Tool[1]:GUN C1 Base[1]:Actros ;%{PE}%R 4.1.16,%MKUKATPBASIS,%CMOVE,%VPTP,%P 1:PTP, 2:p1088, 3:C_PTP, 5:50, 7:P_OLP62
$BWDSTART = FALSE
PDAT_ACT=PP_OLP62
BAS(#PTP_DAT)
FDAT_ACT=Fp1088
BAS(#FRAMES)
BAS(#VEL_PTP,50)
PTP Xp1088 C_PTP
;ENDFOLD

;FOLD ; SWP_60_5208;%{PE}%R2.2,%MKUKATPBASIS,%CCOMMENT,%VNORMAL,%P 2: SWP_60_5208
;ENDFOLD
;FOLD PTP swp_60_5208 PDAT43 SPOT Gun= 1 RETR CLS PgNo1= 86 ACTIVE= 1 Tool[1]:GUN C1 Base[1]:Actros ;%{PE}%R 4.1.12,%MKUKATPSPOT,%CSPOT,%VPTP,%P 1:PTP, 2:swp_60_5208, 3:, 5:100, 7:PDAT43, 10:1, 12:#FIRST, 14:#CLO, 16:86, 18:1, 20:0, 22:0, 24:1, 25:NORMAL
$BWDSTART = FALSE
PDAT_ACT=PPDAT43
BAS(#PTP_DAT)
FDAT_ACT=Fswp_60_5208
BAS(#FRAMES)
BAS(#VEL_PTP,PPDAT43.VEL)
S_ACT.GUN=1
S_ACT.PAIR=SDEFAULT.PAIR
S_ACT.RETR=#CLO
S_ACT.CLO_TM=1
S_ACT.PGNO1=86
S_ACT.PGNO2=SDEFAULT.PGNO2
S_ACT.PRESS1=SDEFAULT.PRESS1
S_ACT.PRESS2=SDEFAULT.PRESS2
S_READY=FALSE
PTP Xswp_60_5208
USERSPOT(#SPOT, S_ACT)
WAIT FOR S_READY
;ENDFOLD

;FOLD ; SWP_60_5207;%{PE}%R2.2,%MKUKATPBASIS,%CCOMMENT,%VNORMAL,%P 2: SWP_60_5207
;ENDFOLD
;FOLD PTP swp_60_5207 PDAT44 SPOT Gun= 1 RETR CLS PgNo1= 87 ACTIVE= 1 Tool[1]:GUN C1 Base[1]:Actros ;%{PE}%R 4.1.12,%MKUKATPSPOT,%CSPOT,%VPTP,%P 1:PTP, 2:swp_60_5207, 3:, 5:100, 7:PDAT44, 10:1, 12:#FIRST, 14:#CLO, 16:87, 18:1, 20:0, 22:0, 24:1, 25:NORMAL
$BWDSTART = FALSE
PDAT_ACT=PPDAT44
BAS(#PTP_DAT)
FDAT_ACT=Fswp_60_5207
BAS(#FRAMES)
BAS(#VEL_PTP,PPDAT44.VEL)
S_ACT.GUN=1
S_ACT.PAIR=SDEFAULT.PAIR
S_ACT.RETR=#CLO
S_ACT.CLO_TM=1
S_ACT.PGNO1=87
S_ACT.PGNO2=SDEFAULT.PGNO2
S_ACT.PRESS1=SDEFAULT.PRESS1
S_ACT.PRESS2=SDEFAULT.PRESS2
S_READY=FALSE
PTP Xswp_60_5207
USERSPOT(#SPOT, S_ACT)
WAIT FOR S_READY
;ENDFOLD

;FOLD ;  SWP_60_5206;%{PE}%R 4.1.16,%MKUKATPBASIS,%CCOMMENT,%VNORMAL,%P 2: SWP_60_5206
;ENDFOLD
;FOLD PTP SWP_60_5206 PDAT78 SPOT Gun= 1 RETR CLS PgNo1= 130 ACTIVE= 1 Tool[1]:GUN C1 Base[1]:Actros ;%{PE}%R 4.1.12,%MKUKATPSPOT,%CSPOT,%VPTP,%P 1:PTP, 2:SWP_60_5206, 3:, 5:70, 7:PDAT78, 10:1, 12:#FIRST, 14:#CLO, 16:130, 18:1, 20:0, 22:0, 24:1, 25:NORMAL
$BWDSTART = FALSE
PDAT_ACT=PPDAT78
BAS(#PTP_DAT)
FDAT_ACT=FSWP_60_5206
BAS(#FRAMES)
BAS(#VEL_PTP,PPDAT78.VEL)
S_ACT.GUN=1
S_ACT.PAIR=SDEFAULT.PAIR
S_ACT.RETR=#CLO
S_ACT.CLO_TM=1
S_ACT.PGNO1=130
S_ACT.PGNO2=SDEFAULT.PGNO2
S_ACT.PRESS1=SDEFAULT.PRESS1
S_ACT.PRESS2=SDEFAULT.PRESS2
S_READY=FALSE
PTP XSWP_60_5206
USERSPOT(#SPOT, S_ACT)
WAIT FOR S_READY
;ENDFOLD

;FOLD ;  SWP_60_5205;%{PE}%R 4.1.16,%MKUKATPBASIS,%CCOMMENT,%VNORMAL,%P 2: SWP_60_5205
;ENDFOLD
;FOLD PTP SWP_60_5205 PDAT79 SPOT Gun= 1 RETR CLS PgNo1= 131 ACTIVE= 1 Tool[1]:GUN C1 Base[1]:Actros ;%{PE}%R 4.1.12,%MKUKATPSPOT,%CSPOT,%VPTP,%P 1:PTP, 2:SWP_60_5205, 3:, 5:70, 7:PDAT79, 10:1, 12:#FIRST, 14:#CLO, 16:131, 18:1, 20:0, 22:0, 24:1, 25:NORMAL
$BWDSTART = FALSE
PDAT_ACT=PPDAT79
BAS(#PTP_DAT)
FDAT_ACT=FSWP_60_5205
BAS(#FRAMES)
BAS(#VEL_PTP,PPDAT79.VEL)
S_ACT.GUN=1
S_ACT.PAIR=SDEFAULT.PAIR
S_ACT.RETR=#CLO
S_ACT.CLO_TM=1
S_ACT.PGNO1=131
S_ACT.PGNO2=SDEFAULT.PGNO2
S_ACT.PRESS1=SDEFAULT.PRESS1
S_ACT.PRESS2=SDEFAULT.PRESS2
S_READY=FALSE
PTP XSWP_60_5205
USERSPOT(#SPOT, S_ACT)
WAIT FOR S_READY
;ENDFOLD

;FOLD ;  SWP_60_5204;%{PE}%R 4.1.16,%MKUKATPBASIS,%CCOMMENT,%VNORMAL,%P 2: SWP_60_5204
;ENDFOLD
;FOLD PTP SWP_60_5204 PDAT80 SPOT Gun= 1 RETR CLS PgNo1= 132 ACTIVE= 1 Tool[1]:GUN C1 Base[1]:Actros ;%{PE}%R 4.1.12,%MKUKATPSPOT,%CSPOT,%VPTP,%P 1:PTP, 2:SWP_60_5204, 3:, 5:70, 7:PDAT80, 10:1, 12:#FIRST, 14:#CLO, 16:132, 18:1, 20:0, 22:0, 24:1, 25:NORMAL
$BWDSTART = FALSE
PDAT_ACT=PPDAT80
BAS(#PTP_DAT)
FDAT_ACT=FSWP_60_5204
BAS(#FRAMES)
BAS(#VEL_PTP,PPDAT80.VEL)
S_ACT.GUN=1
S_ACT.PAIR=SDEFAULT.PAIR
S_ACT.RETR=#CLO
S_ACT.CLO_TM=1
S_ACT.PGNO1=132
S_ACT.PGNO2=SDEFAULT.PGNO2
S_ACT.PRESS1=SDEFAULT.PRESS1
S_ACT.PRESS2=SDEFAULT.PRESS2
S_READY=FALSE
PTP XSWP_60_5204
USERSPOT(#SPOT, S_ACT)
WAIT FOR S_READY
;ENDFOLD


;FOLD ;  SWP_60_5202;%{PE}%R 4.1.16,%MKUKATPBASIS,%CCOMMENT,%VNORMAL,%P 2: SWP_60_5202
;ENDFOLD
;FOLD PTP SWP_60_5202 PDAT81 SPOT Gun= 1 RETR CLS PgNo1= 133 ACTIVE= 1 Tool[1]:GUN C1 Base[1]:Actros ;%{PE}%R 4.1.12,%MKUKATPSPOT,%CSPOT,%VPTP,%P 1:PTP, 2:SWP_60_5202, 3:, 5:70, 7:PDAT81, 10:1, 12:#FIRST, 14:#CLO, 16:133, 18:1, 20:0, 22:0, 24:1, 25:NORMAL
$BWDSTART = FALSE
PDAT_ACT=PPDAT81
BAS(#PTP_DAT)
FDAT_ACT=FSWP_60_5202
BAS(#FRAMES)
BAS(#VEL_PTP,PPDAT81.VEL)
S_ACT.GUN=1
S_ACT.PAIR=SDEFAULT.PAIR
S_ACT.RETR=#CLO
S_ACT.CLO_TM=1
S_ACT.PGNO1=133
S_ACT.PGNO2=SDEFAULT.PGNO2
S_ACT.PRESS1=SDEFAULT.PRESS1
S_ACT.PRESS2=SDEFAULT.PRESS2
S_READY=FALSE
PTP XSWP_60_5202
USERSPOT(#SPOT, S_ACT)
WAIT FOR S_READY
;ENDFOLD

;FOLD ;  SWP_60_5200;%{PE}%R 4.1.16,%MKUKATPBASIS,%CCOMMENT,%VNORMAL,%P 2: SWP_60_5200
;ENDFOLD
;FOLD PTP SWP_60_5200 PDAT82 SPOT Gun= 1 RETR CLS PgNo1= 134 ACTIVE= 1 Tool[1]:GUN C1 Base[1]:Actros ;%{PE}%R 4.1.12,%MKUKATPSPOT,%CSPOT,%VPTP,%P 1:PTP, 2:SWP_60_5200, 3:, 5:70, 7:PDAT82, 10:1, 12:#FIRST, 14:#CLO, 16:134, 18:1, 20:0, 22:0, 24:1, 25:NORMAL
$BWDSTART = FALSE
PDAT_ACT=PPDAT82
BAS(#PTP_DAT)
FDAT_ACT=FSWP_60_5200
BAS(#FRAMES)
BAS(#VEL_PTP,PPDAT82.VEL)
S_ACT.GUN=1
S_ACT.PAIR=SDEFAULT.PAIR
S_ACT.RETR=#CLO
S_ACT.CLO_TM=1
S_ACT.PGNO1=134
S_ACT.PGNO2=SDEFAULT.PGNO2
S_ACT.PRESS1=SDEFAULT.PRESS1
S_ACT.PRESS2=SDEFAULT.PRESS2
S_READY=FALSE
PTP XSWP_60_5200
USERSPOT(#SPOT, S_ACT)
WAIT FOR S_READY
;ENDFOLD

;FOLD ; SWP_60_5201;%{PE}%R2.2,%MKUKATPBASIS,%CCOMMENT,%VNORMAL,%P 2: SWP_60_5201
;ENDFOLD
;FOLD PTP swp_60_5201 PDAT45 SPOT Gun= 1 RETR CLS PgNo1= 88 ACTIVE= 1 Tool[1]:GUN C1 Base[1]:Actros ;%{PE}%R 4.1.12,%MKUKATPSPOT,%CSPOT,%VPTP,%P 1:PTP, 2:swp_60_5201, 3:, 5:100, 7:PDAT45, 10:1, 12:#FIRST, 14:#CLO, 16:88, 18:1, 20:0, 22:0, 24:1, 25:NORMAL
$BWDSTART = FALSE
PDAT_ACT=PPDAT45
BAS(#PTP_DAT)
FDAT_ACT=Fswp_60_5201
BAS(#FRAMES)
BAS(#VEL_PTP,PPDAT45.VEL)
S_ACT.GUN=1
S_ACT.PAIR=SDEFAULT.PAIR
S_ACT.RETR=#CLO
S_ACT.CLO_TM=1
S_ACT.PGNO1=88
S_ACT.PGNO2=SDEFAULT.PGNO2
S_ACT.PRESS1=SDEFAULT.PRESS1
S_ACT.PRESS2=SDEFAULT.PRESS2
S_READY=FALSE
PTP Xswp_60_5201
USERSPOT(#SPOT, S_ACT)
WAIT FOR S_READY
;ENDFOLD

;FOLD Kollision.Ueberwachung_3_Ein ;%{PE}%MKUKATPUSER
COLLSTOP( 3, 1 ) ;INTERRUPTUEBERWACHT
;ENDFOLD

;FOLD ; SWP_60_5199;%{PE}%R2.2,%MKUKATPBASIS,%CCOMMENT,%VNORMAL,%P 2: SWP_60_5199
;ENDFOLD
;FOLD PTP swp_60_5199 PDAT46 SPOT Gun= 1 RETR CLS PgNo1= 89 ACTIVE= 1 Tool[1]:GUN C1 Base[1]:Actros ;%{PE}%R 4.1.12,%MKUKATPSPOT,%CSPOT,%VPTP,%P 1:PTP, 2:swp_60_5199, 3:, 5:100, 7:PDAT46, 10:1, 12:#FIRST, 14:#CLO, 16:89, 18:1, 20:0, 22:0, 24:1, 25:NORMAL
$BWDSTART = FALSE
PDAT_ACT=PPDAT46
BAS(#PTP_DAT)
FDAT_ACT=Fswp_60_5199
BAS(#FRAMES)
BAS(#VEL_PTP,PPDAT46.VEL)
S_ACT.GUN=1
S_ACT.PAIR=SDEFAULT.PAIR
S_ACT.RETR=#CLO
S_ACT.CLO_TM=1
S_ACT.PGNO1=89
S_ACT.PGNO2=SDEFAULT.PGNO2
S_ACT.PRESS1=SDEFAULT.PRESS1
S_ACT.PRESS2=SDEFAULT.PRESS2
S_READY=FALSE
PTP Xswp_60_5199
USERSPOT(#SPOT, S_ACT)
WAIT FOR S_READY
;ENDFOLD

;FOLD ;  SWP_60_5198;%{PE}%R 4.1.16,%MKUKATPBASIS,%CCOMMENT,%VNORMAL,%P 2: SWP_60_5198
;ENDFOLD
;FOLD PTP SWP_60_5198 PDAT83 SPOT Gun= 1 RETR CLS PgNo1= 135 ACTIVE= 1 Tool[1]:GUN C1 Base[1]:Actros ;%{PE}%R 4.1.12,%MKUKATPSPOT,%CSPOT,%VPTP,%P 1:PTP, 2:SWP_60_5198, 3:, 5:70, 7:PDAT83, 10:1, 12:#FIRST, 14:#CLO, 16:135, 18:1, 20:0, 22:0, 24:1, 25:NORMAL
$BWDSTART = FALSE
PDAT_ACT=PPDAT83
BAS(#PTP_DAT)
FDAT_ACT=FSWP_60_5198
BAS(#FRAMES)
BAS(#VEL_PTP,PPDAT83.VEL)
S_ACT.GUN=1
S_ACT.PAIR=SDEFAULT.PAIR
S_ACT.RETR=#CLO
S_ACT.CLO_TM=1
S_ACT.PGNO1=135
S_ACT.PGNO2=SDEFAULT.PGNO2
S_ACT.PRESS1=SDEFAULT.PRESS1
S_ACT.PRESS2=SDEFAULT.PRESS2
S_READY=FALSE
PTP XSWP_60_5198
USERSPOT(#SPOT, S_ACT)
WAIT FOR S_READY
;ENDFOLD

;FOLD ; SWP_60_5197;%{PE}%R2.2,%MKUKATPBASIS,%CCOMMENT,%VNORMAL,%P 2: SWP_60_5197
;ENDFOLD
;FOLD PTP swp_60_5197 PDAT47 SPOT Gun= 1 RETR CLS PgNo1= 90 ACTIVE= 1 Tool[1]:GUN C1 Base[1]:Actros ;%{PE}%R 4.1.12,%MKUKATPSPOT,%CSPOT,%VPTP,%P 1:PTP, 2:swp_60_5197, 3:, 5:100, 7:PDAT47, 10:1, 12:#FIRST, 14:#CLO, 16:90, 18:1, 20:0, 22:0, 24:1, 25:NORMAL
$BWDSTART = FALSE
PDAT_ACT=PPDAT47
BAS(#PTP_DAT)
FDAT_ACT=Fswp_60_5197
BAS(#FRAMES)
BAS(#VEL_PTP,PPDAT47.VEL)
S_ACT.GUN=1
S_ACT.PAIR=SDEFAULT.PAIR
S_ACT.RETR=#CLO
S_ACT.CLO_TM=1
S_ACT.PGNO1=90
S_ACT.PGNO2=SDEFAULT.PGNO2
S_ACT.PRESS1=SDEFAULT.PRESS1
S_ACT.PRESS2=SDEFAULT.PRESS2
S_READY=FALSE
PTP Xswp_60_5197
USERSPOT(#SPOT, S_ACT)
WAIT FOR S_READY
;ENDFOLD

;FOLD ;  SWP_60_5196;%{PE}%R 4.1.16,%MKUKATPBASIS,%CCOMMENT,%VNORMAL,%P 2: SWP_60_5196
;ENDFOLD
;FOLD PTP SWP_60_5196 PDAT84 SPOT Gun= 1 RETR CLS PgNo1= 136 ACTIVE= 1 Tool[1]:GUN C1 Base[1]:Actros ;%{PE}%R 4.1.12,%MKUKATPSPOT,%CSPOT,%VPTP,%P 1:PTP, 2:SWP_60_5196, 3:, 5:70, 7:PDAT84, 10:1, 12:#FIRST, 14:#CLO, 16:136, 18:1, 20:0, 22:0, 24:1, 25:NORMAL
$BWDSTART = FALSE
PDAT_ACT=PPDAT84
BAS(#PTP_DAT)
FDAT_ACT=FSWP_60_5196
BAS(#FRAMES)
BAS(#VEL_PTP,PPDAT84.VEL)
S_ACT.GUN=1
S_ACT.PAIR=SDEFAULT.PAIR
S_ACT.RETR=#CLO
S_ACT.CLO_TM=1
S_ACT.PGNO1=136
S_ACT.PGNO2=SDEFAULT.PGNO2
S_ACT.PRESS1=SDEFAULT.PRESS1
S_ACT.PRESS2=SDEFAULT.PRESS2
S_READY=FALSE
PTP XSWP_60_5196
USERSPOT(#SPOT, S_ACT)
WAIT FOR S_READY
;ENDFOLD

;FOLD PTP SWP_60_5203 CONT Vel= 65 % PDAT85 Tool[1]:GUN C1 Base[1]:Actros ;%{PE}%R 4.1.16,%MKUKATPBASIS,%CMOVE,%VPTP,%P 1:PTP, 2:SWP_60_5203, 3:C_PTP, 5:65, 7:PDAT85
$BWDSTART = FALSE
PDAT_ACT=PPDAT85
BAS(#PTP_DAT)
FDAT_ACT=FSWP_60_5203
BAS(#FRAMES)
BAS(#VEL_PTP,65)
PTP XSWP_60_5203 C_PTP
;ENDFOLD

;FOLD ;  SWP_60_5194;%{PE}%R 4.1.16,%MKUKATPBASIS,%CCOMMENT,%VNORMAL,%P 2: SWP_60_5194
;ENDFOLD
;FOLD PTP SWP_60_5194 PDAT86 SPOT Gun= 1 RETR CLS PgNo1= 137 ACTIVE= 1 Tool[1]:GUN C1 Base[1]:Actros ;%{PE}%R 4.1.12,%MKUKATPSPOT,%CSPOT,%VPTP,%P 1:PTP, 2:SWP_60_5194, 3:, 5:80, 7:PDAT86, 10:1, 12:#FIRST, 14:#CLO, 16:137, 18:1, 20:0, 22:0, 24:1, 25:NORMAL
$BWDSTART = FALSE
PDAT_ACT=PPDAT86
BAS(#PTP_DAT)
FDAT_ACT=FSWP_60_5194
BAS(#FRAMES)
BAS(#VEL_PTP,PPDAT86.VEL)
S_ACT.GUN=1
S_ACT.PAIR=SDEFAULT.PAIR
S_ACT.RETR=#CLO
S_ACT.CLO_TM=1
S_ACT.PGNO1=137
S_ACT.PGNO2=SDEFAULT.PGNO2
S_ACT.PRESS1=SDEFAULT.PRESS1
S_ACT.PRESS2=SDEFAULT.PRESS2
S_READY=FALSE
PTP XSWP_60_5194
USERSPOT(#SPOT, S_ACT)
WAIT FOR S_READY
;ENDFOLD

;FOLD ;  SWP_60_5193;%{PE}%R 4.1.16,%MKUKATPBASIS,%CCOMMENT,%VNORMAL,%P 2: SWP_60_5193
;ENDFOLD
;FOLD PTP SWP_60_5193 PDAT87 SPOT Gun= 1 RETR CLS PgNo1= 138 ACTIVE= 1 Tool[1]:GUN C1 Base[1]:Actros ;%{PE}%R 4.1.12,%MKUKATPSPOT,%CSPOT,%VPTP,%P 1:PTP, 2:SWP_60_5193, 3:, 5:80, 7:PDAT87, 10:1, 12:#FIRST, 14:#CLO, 16:138, 18:1, 20:0, 22:0, 24:1, 25:NORMAL
$BWDSTART = FALSE
PDAT_ACT=PPDAT87
BAS(#PTP_DAT)
FDAT_ACT=FSWP_60_5193
BAS(#FRAMES)
BAS(#VEL_PTP,PPDAT87.VEL)
S_ACT.GUN=1
S_ACT.PAIR=SDEFAULT.PAIR
S_ACT.RETR=#CLO
S_ACT.CLO_TM=1
S_ACT.PGNO1=138
S_ACT.PGNO2=SDEFAULT.PGNO2
S_ACT.PRESS1=SDEFAULT.PRESS1
S_ACT.PRESS2=SDEFAULT.PRESS2
S_READY=FALSE
PTP XSWP_60_5193
USERSPOT(#SPOT, S_ACT)
WAIT FOR S_READY
;ENDFOLD

;FOLD ;  SWP_60_5192;%{PE}%R 4.1.16,%MKUKATPBASIS,%CCOMMENT,%VNORMAL,%P 2: SWP_60_5192
;ENDFOLD
;FOLD PTP SWP_60_5192 PDAT88 SPOT Gun= 1 RETR CLS PgNo1= 139 ACTIVE= 1 Tool[1]:GUN C1 Base[1]:Actros ;%{PE}%R 4.1.12,%MKUKATPSPOT,%CSPOT,%VPTP,%P 1:PTP, 2:SWP_60_5192, 3:, 5:80, 7:PDAT88, 10:1, 12:#FIRST, 14:#CLO, 16:139, 18:1, 20:0, 22:0, 24:1, 25:NORMAL
$BWDSTART = FALSE
PDAT_ACT=PPDAT88
BAS(#PTP_DAT)
FDAT_ACT=FSWP_60_5192
BAS(#FRAMES)
BAS(#VEL_PTP,PPDAT88.VEL)
S_ACT.GUN=1
S_ACT.PAIR=SDEFAULT.PAIR
S_ACT.RETR=#CLO
S_ACT.CLO_TM=1
S_ACT.PGNO1=139
S_ACT.PGNO2=SDEFAULT.PGNO2
S_ACT.PRESS1=SDEFAULT.PRESS1
S_ACT.PRESS2=SDEFAULT.PRESS2
S_READY=FALSE
PTP XSWP_60_5192
USERSPOT(#SPOT, S_ACT)
WAIT FOR S_READY
;ENDFOLD

;FOLD PTP SWP_60_5195 CONT Vel= 65 % PDAT89 Tool[1]:GUN C1 Base[1]:Actros ;%{PE}%R 4.1.16,%MKUKATPBASIS,%CMOVE,%VPTP,%P 1:PTP, 2:SWP_60_5195, 3:C_PTP, 5:65, 7:PDAT89
$BWDSTART = FALSE
PDAT_ACT=PPDAT89
BAS(#PTP_DAT)
FDAT_ACT=FSWP_60_5195
BAS(#FRAMES)
BAS(#VEL_PTP,65)
PTP XSWP_60_5195 C_PTP
;ENDFOLD
;FOLD PTP p1095 CONT Vel= 65 % P_OLP69 Tool[1]:GUN C1 Base[1]:Actros ;%{PE}%R 4.1.16,%MKUKATPBASIS,%CMOVE,%VPTP,%P 1:PTP, 2:p1095, 3:C_PTP, 5:65, 7:P_OLP69
$BWDSTART = FALSE
PDAT_ACT=PP_OLP69
BAS(#PTP_DAT)
FDAT_ACT=Fp1095
BAS(#FRAMES)
BAS(#VEL_PTP,65)
PTP Xp1095 C_PTP
;ENDFOLD
;FOLD PTP p1096 CONT Vel= 65 % P_OLP70 Tool[1]:GUN C1 Base[1]:Actros ;%{PE}%R 4.1.16,%MKUKATPBASIS,%CMOVE,%VPTP,%P 1:PTP, 2:p1096, 3:C_PTP, 5:65, 7:P_OLP70
$BWDSTART = FALSE
PDAT_ACT=PP_OLP70
BAS(#PTP_DAT)
FDAT_ACT=Fp1096
BAS(#FRAMES)
BAS(#VEL_PTP,65)
PTP Xp1096 C_PTP
;ENDFOLD
;FOLD PTP p1097 CONT Vel= 50 % P_OLP71 Tool[1]:GUN C1 Base[1]:Actros ;%{PE}%R 4.1.16,%MKUKATPBASIS,%CMOVE,%VPTP,%P 1:PTP, 2:p1097, 3:C_PTP, 5:50, 7:P_OLP71
$BWDSTART = FALSE
PDAT_ACT=PP_OLP71
BAS(#PTP_DAT)
FDAT_ACT=Fp1097
BAS(#FRAMES)
BAS(#VEL_PTP,50)
PTP Xp1097 C_PTP
;ENDFOLD

;FOLD ; SWP_60_5225;%{PE}%R2.2,%MKUKATPBASIS,%CCOMMENT,%VNORMAL,%P 2: SWP_60_5225
;ENDFOLD
;FOLD PTP swp_60_5225 PDAT48 SPOT Gun= 1 RETR CLS PgNo1= 91 ACTIVE= 1 Tool[1]:GUN C1 Base[1]:Actros ;%{PE}%R 4.1.12,%MKUKATPSPOT,%CSPOT,%VPTP,%P 1:PTP, 2:swp_60_5225, 3:, 5:100, 7:PDAT48, 10:1, 12:#FIRST, 14:#CLO, 16:91, 18:1, 20:0, 22:0, 24:1, 25:NORMAL
$BWDSTART = FALSE
PDAT_ACT=PPDAT48
BAS(#PTP_DAT)
FDAT_ACT=Fswp_60_5225
BAS(#FRAMES)
BAS(#VEL_PTP,PPDAT48.VEL)
S_ACT.GUN=1
S_ACT.PAIR=SDEFAULT.PAIR
S_ACT.RETR=#CLO
S_ACT.CLO_TM=1
S_ACT.PGNO1=91
S_ACT.PGNO2=SDEFAULT.PGNO2
S_ACT.PRESS1=SDEFAULT.PRESS1
S_ACT.PRESS2=SDEFAULT.PRESS2
S_READY=FALSE
PTP Xswp_60_5225
USERSPOT(#SPOT, S_ACT)
WAIT FOR S_READY
;ENDFOLD

;FOLD ; SWP_60_5224;%{PE}%R2.2,%MKUKATPBASIS,%CCOMMENT,%VNORMAL,%P 2: SWP_60_5224
;ENDFOLD
;FOLD PTP swp_60_5224 PDAT49 SPOT Gun= 1 RETR CLS PgNo1= 92 ACTIVE= 1 Tool[1]:GUN C1 Base[1]:Actros ;%{PE}%R 4.1.12,%MKUKATPSPOT,%CSPOT,%VPTP,%P 1:PTP, 2:swp_60_5224, 3:, 5:100, 7:PDAT49, 10:1, 12:#FIRST, 14:#CLO, 16:92, 18:1, 20:0, 22:0, 24:1, 25:NORMAL
$BWDSTART = FALSE
PDAT_ACT=PPDAT49
BAS(#PTP_DAT)
FDAT_ACT=Fswp_60_5224
BAS(#FRAMES)
BAS(#VEL_PTP,PPDAT49.VEL)
S_ACT.GUN=1
S_ACT.PAIR=SDEFAULT.PAIR
S_ACT.RETR=#CLO
S_ACT.CLO_TM=1
S_ACT.PGNO1=92
S_ACT.PGNO2=SDEFAULT.PGNO2
S_ACT.PRESS1=SDEFAULT.PRESS1
S_ACT.PRESS2=SDEFAULT.PRESS2
S_READY=FALSE
PTP Xswp_60_5224
USERSPOT(#SPOT, S_ACT)
WAIT FOR S_READY
;ENDFOLD

;FOLD ; SWP_60_5223;%{PE}%R2.2,%MKUKATPBASIS,%CCOMMENT,%VNORMAL,%P 2: SWP_60_5223
;ENDFOLD
;FOLD PTP swp_60_5223 PDAT50 SPOT Gun= 1 RETR CLS PgNo1= 93 ACTIVE= 1 Tool[1]:GUN C1 Base[1]:Actros ;%{PE}%R 4.1.12,%MKUKATPSPOT,%CSPOT,%VPTP,%P 1:PTP, 2:swp_60_5223, 3:, 5:100, 7:PDAT50, 10:1, 12:#FIRST, 14:#CLO, 16:93, 18:1, 20:0, 22:0, 24:1, 25:NORMAL
$BWDSTART = FALSE
PDAT_ACT=PPDAT50
BAS(#PTP_DAT)
FDAT_ACT=Fswp_60_5223
BAS(#FRAMES)
BAS(#VEL_PTP,PPDAT50.VEL)
S_ACT.GUN=1
S_ACT.PAIR=SDEFAULT.PAIR
S_ACT.RETR=#CLO
S_ACT.CLO_TM=1
S_ACT.PGNO1=93
S_ACT.PGNO2=SDEFAULT.PGNO2
S_ACT.PRESS1=SDEFAULT.PRESS1
S_ACT.PRESS2=SDEFAULT.PRESS2
S_READY=FALSE
PTP Xswp_60_5223
USERSPOT(#SPOT, S_ACT)
WAIT FOR S_READY
;ENDFOLD

;FOLD PTP p1101 CONT Vel= 50 % P_OLP75 Tool[1]:GUN C1 Base[1]:Actros ;%{PE}%R 4.1.16,%MKUKATPBASIS,%CMOVE,%VPTP,%P 1:PTP, 2:p1101, 3:C_PTP, 5:50, 7:P_OLP75
$BWDSTART = FALSE
PDAT_ACT=PP_OLP75
BAS(#PTP_DAT)
FDAT_ACT=Fp1101
BAS(#FRAMES)
BAS(#VEL_PTP,50)
PTP Xp1101 C_PTP
;ENDFOLD

;FOLD ; SWP_60_5222;%{PE}%R2.2,%MKUKATPBASIS,%CCOMMENT,%VNORMAL,%P 2: SWP_60_5222
;ENDFOLD
;FOLD PTP swp_60_5222 PDAT51 SPOT Gun= 1 RETR CLS PgNo1= 94 ACTIVE= 1 Tool[1]:GUN C1 Base[1]:Actros ;%{PE}%R 4.1.12,%MKUKATPSPOT,%CSPOT,%VPTP,%P 1:PTP, 2:swp_60_5222, 3:, 5:100, 7:PDAT51, 10:1, 12:#FIRST, 14:#CLO, 16:94, 18:1, 20:0, 22:0, 24:1, 25:NORMAL
$BWDSTART = FALSE
PDAT_ACT=PPDAT51
BAS(#PTP_DAT)
FDAT_ACT=Fswp_60_5222
BAS(#FRAMES)
BAS(#VEL_PTP,PPDAT51.VEL)
S_ACT.GUN=1
S_ACT.PAIR=SDEFAULT.PAIR
S_ACT.RETR=#CLO
S_ACT.CLO_TM=1
S_ACT.PGNO1=94
S_ACT.PGNO2=SDEFAULT.PGNO2
S_ACT.PRESS1=SDEFAULT.PRESS1
S_ACT.PRESS2=SDEFAULT.PRESS2
S_READY=FALSE
PTP Xswp_60_5222
USERSPOT(#SPOT, S_ACT)
WAIT FOR S_READY
;ENDFOLD

;FOLD ; SWP_60_5221;%{PE}%R2.2,%MKUKATPBASIS,%CCOMMENT,%VNORMAL,%P 2: SWP_60_5221
;ENDFOLD
;FOLD PTP swp_60_5221 PDAT52 SPOT Gun= 1 RETR CLS PgNo1= 95 ACTIVE= 1 Tool[1]:GUN C1 Base[1]:Actros ;%{PE}%R 4.1.12,%MKUKATPSPOT,%CSPOT,%VPTP,%P 1:PTP, 2:swp_60_5221, 3:, 5:100, 7:PDAT52, 10:1, 12:#FIRST, 14:#CLO, 16:95, 18:1, 20:0, 22:0, 24:1, 25:NORMAL
$BWDSTART = FALSE
PDAT_ACT=PPDAT52
BAS(#PTP_DAT)
FDAT_ACT=Fswp_60_5221
BAS(#FRAMES)
BAS(#VEL_PTP,PPDAT52.VEL)
S_ACT.GUN=1
S_ACT.PAIR=SDEFAULT.PAIR
S_ACT.RETR=#CLO
S_ACT.CLO_TM=1
S_ACT.PGNO1=95
S_ACT.PGNO2=SDEFAULT.PGNO2
S_ACT.PRESS1=SDEFAULT.PRESS1
S_ACT.PRESS2=SDEFAULT.PRESS2
S_READY=FALSE
PTP Xswp_60_5221
USERSPOT(#SPOT, S_ACT)
WAIT FOR S_READY
;ENDFOLD

;FOLD ; SWP_60_5220;%{PE}%R2.2,%MKUKATPBASIS,%CCOMMENT,%VNORMAL,%P 2: SWP_60_5220
;ENDFOLD
;FOLD PTP swp_60_5220 PDAT53 SPOT Gun= 1 RETR CLS PgNo1= 96 ACTIVE= 1 Tool[1]:GUN C1 Base[1]:Actros ;%{PE}%R 4.1.12,%MKUKATPSPOT,%CSPOT,%VPTP,%P 1:PTP, 2:swp_60_5220, 3:, 5:100, 7:PDAT53, 10:1, 12:#FIRST, 14:#CLO, 16:96, 18:1, 20:0, 22:0, 24:1, 25:NORMAL
$BWDSTART = FALSE
PDAT_ACT=PPDAT53
BAS(#PTP_DAT)
FDAT_ACT=Fswp_60_5220
BAS(#FRAMES)
BAS(#VEL_PTP,PPDAT53.VEL)
S_ACT.GUN=1
S_ACT.PAIR=SDEFAULT.PAIR
S_ACT.RETR=#CLO
S_ACT.CLO_TM=1
S_ACT.PGNO1=96
S_ACT.PGNO2=SDEFAULT.PGNO2
S_ACT.PRESS1=SDEFAULT.PRESS1
S_ACT.PRESS2=SDEFAULT.PRESS2
S_READY=FALSE
PTP Xswp_60_5220
USERSPOT(#SPOT, S_ACT)
WAIT FOR S_READY
;ENDFOLD

;FOLD PTP p1105 CONT Vel= 50 % P_OLP79 Tool[1]:GUN C1 Base[1]:Actros ;%{PE}%R 4.1.16,%MKUKATPBASIS,%CMOVE,%VPTP,%P 1:PTP, 2:p1105, 3:C_PTP, 5:50, 7:P_OLP79
$BWDSTART = FALSE
PDAT_ACT=PP_OLP79
BAS(#PTP_DAT)
FDAT_ACT=Fp1105
BAS(#FRAMES)
BAS(#VEL_PTP,50)
PTP Xp1105 C_PTP
;ENDFOLD

;FOLD ; SWP_60_5239;%{PE}%R2.2,%MKUKATPBASIS,%CCOMMENT,%VNORMAL,%P 2: SWP_60_5239
;ENDFOLD
;FOLD PTP swp_60_5239 PDAT54 SPOT Gun= 1 RETR CLS PgNo1= 97 ACTIVE= 1 Tool[1]:GUN C1 Base[1]:Actros ;%{PE}%R 4.1.12,%MKUKATPSPOT,%CSPOT,%VPTP,%P 1:PTP, 2:swp_60_5239, 3:, 5:100, 7:PDAT54, 10:1, 12:#FIRST, 14:#CLO, 16:97, 18:1, 20:0, 22:0, 24:1, 25:NORMAL
$BWDSTART = FALSE
PDAT_ACT=PPDAT54
BAS(#PTP_DAT)
FDAT_ACT=Fswp_60_5239
BAS(#FRAMES)
BAS(#VEL_PTP,PPDAT54.VEL)
S_ACT.GUN=1
S_ACT.PAIR=SDEFAULT.PAIR
S_ACT.RETR=#CLO
S_ACT.CLO_TM=1
S_ACT.PGNO1=97
S_ACT.PGNO2=SDEFAULT.PGNO2
S_ACT.PRESS1=SDEFAULT.PRESS1
S_ACT.PRESS2=SDEFAULT.PRESS2
S_READY=FALSE
PTP Xswp_60_5239
USERSPOT(#SPOT, S_ACT)
WAIT FOR S_READY
;ENDFOLD

;FOLD ; SWP_60_5238;%{PE}%R2.2,%MKUKATPBASIS,%CCOMMENT,%VNORMAL,%P 2: SWP_60_5238
;ENDFOLD
;FOLD PTP swp_60_5238 PDAT55 SPOT Gun= 1 RETR CLS PgNo1= 98 ACTIVE= 1 Tool[1]:GUN C1 Base[1]:Actros ;%{PE}%R 4.1.12,%MKUKATPSPOT,%CSPOT,%VPTP,%P 1:PTP, 2:swp_60_5238, 3:, 5:100, 7:PDAT55, 10:1, 12:#FIRST, 14:#CLO, 16:98, 18:1, 20:0, 22:0, 24:1, 25:NORMAL
$BWDSTART = FALSE
PDAT_ACT=PPDAT55
BAS(#PTP_DAT)
FDAT_ACT=Fswp_60_5238
BAS(#FRAMES)
BAS(#VEL_PTP,PPDAT55.VEL)
S_ACT.GUN=1
S_ACT.PAIR=SDEFAULT.PAIR
S_ACT.RETR=#CLO
S_ACT.CLO_TM=1
S_ACT.PGNO1=98
S_ACT.PGNO2=SDEFAULT.PGNO2
S_ACT.PRESS1=SDEFAULT.PRESS1
S_ACT.PRESS2=SDEFAULT.PRESS2
S_READY=FALSE
PTP Xswp_60_5238
USERSPOT(#SPOT, S_ACT)
WAIT FOR S_READY
;ENDFOLD

;FOLD ; SWP_60_5237;%{PE}%R2.2,%MKUKATPBASIS,%CCOMMENT,%VNORMAL,%P 2: SWP_60_5237
;ENDFOLD
;FOLD PTP swp_60_5237 PDAT56 SPOT Gun= 1 RETR CLS PgNo1= 99 ACTIVE= 1 Tool[1]:GUN C1 Base[1]:Actros ;%{PE}%R 4.1.12,%MKUKATPSPOT,%CSPOT,%VPTP,%P 1:PTP, 2:swp_60_5237, 3:, 5:100, 7:PDAT56, 10:1, 12:#FIRST, 14:#CLO, 16:99, 18:1, 20:0, 22:0, 24:1, 25:NORMAL
$BWDSTART = FALSE
PDAT_ACT=PPDAT56
BAS(#PTP_DAT)
FDAT_ACT=Fswp_60_5237
BAS(#FRAMES)
BAS(#VEL_PTP,PPDAT56.VEL)
S_ACT.GUN=1
S_ACT.PAIR=SDEFAULT.PAIR
S_ACT.RETR=#CLO
S_ACT.CLO_TM=1
S_ACT.PGNO1=99
S_ACT.PGNO2=SDEFAULT.PGNO2
S_ACT.PRESS1=SDEFAULT.PRESS1
S_ACT.PRESS2=SDEFAULT.PRESS2
S_READY=FALSE
PTP Xswp_60_5237
USERSPOT(#SPOT, S_ACT)
WAIT FOR S_READY
;ENDFOLD

;FOLD PTP p1109 CONT Vel= 50 % P_OLP83 Tool[1]:GUN C1 Base[1]:Actros ;%{PE}%R 4.1.16,%MKUKATPBASIS,%CMOVE,%VPTP,%P 1:PTP, 2:p1109, 3:C_PTP, 5:50, 7:P_OLP83
$BWDSTART = FALSE
PDAT_ACT=PP_OLP83
BAS(#PTP_DAT)
FDAT_ACT=Fp1109
BAS(#FRAMES)
BAS(#VEL_PTP,50)
PTP Xp1109 C_PTP
;ENDFOLD
;FOLD PTP p1110 CONT Vel= 65 % P_OLP84 Tool[1]:GUN C1 Base[1]:Actros ;%{PE}%R 4.1.16,%MKUKATPBASIS,%CMOVE,%VPTP,%P 1:PTP, 2:p1110, 3:C_PTP, 5:65, 7:P_OLP84
$BWDSTART = FALSE
PDAT_ACT=PP_OLP84
BAS(#PTP_DAT)
FDAT_ACT=Fp1110
BAS(#FRAMES)
BAS(#VEL_PTP,65)
PTP Xp1110 C_PTP
;ENDFOLD
;FOLD PTP p1111 CONT Vel= 65 % P_OLP85 Tool[1]:GUN C1 Base[1]:Actros ;%{PE}%R 4.1.16,%MKUKATPBASIS,%CMOVE,%VPTP,%P 1:PTP, 2:p1111, 3:C_PTP, 5:65, 7:P_OLP85
$BWDSTART = FALSE
PDAT_ACT=PP_OLP85
BAS(#PTP_DAT)
FDAT_ACT=Fp1111
BAS(#FRAMES)
BAS(#VEL_PTP,65)
PTP Xp1111 C_PTP
;ENDFOLD
;FOLD PTP p1112 CONT Vel= 50 % P_OLP86 Tool[1]:GUN C1 Base[1]:Actros ;%{PE}%R 4.1.16,%MKUKATPBASIS,%CMOVE,%VPTP,%P 1:PTP, 2:p1112, 3:C_PTP, 5:50, 7:P_OLP86
$BWDSTART = FALSE
PDAT_ACT=PP_OLP86
BAS(#PTP_DAT)
FDAT_ACT=Fp1112
BAS(#FRAMES)
BAS(#VEL_PTP,50)
PTP Xp1112 C_PTP
;ENDFOLD

;FOLD ; SWP_60_5108;%{PE}%R2.2,%MKUKATPBASIS,%CCOMMENT,%VNORMAL,%P 2: SWP_60_5108
;ENDFOLD
;FOLD PTP swp_60_5108 PDAT57 SPOT Gun= 1 RETR CLS PgNo1= 100 ACTIVE= 1 Tool[1]:GUN C1 Base[1]:Actros ;%{PE}%R 4.1.12,%MKUKATPSPOT,%CSPOT,%VPTP,%P 1:PTP, 2:swp_60_5108, 3:, 5:100, 7:PDAT57, 10:1, 12:#FIRST, 14:#CLO, 16:100, 18:1, 20:0, 22:0, 24:1, 25:NORMAL
$BWDSTART = FALSE
PDAT_ACT=PPDAT57
BAS(#PTP_DAT)
FDAT_ACT=Fswp_60_5108
BAS(#FRAMES)
BAS(#VEL_PTP,PPDAT57.VEL)
S_ACT.GUN=1
S_ACT.PAIR=SDEFAULT.PAIR
S_ACT.RETR=#CLO
S_ACT.CLO_TM=1
S_ACT.PGNO1=100
S_ACT.PGNO2=SDEFAULT.PGNO2
S_ACT.PRESS1=SDEFAULT.PRESS1
S_ACT.PRESS2=SDEFAULT.PRESS2
S_READY=FALSE
PTP Xswp_60_5108
USERSPOT(#SPOT, S_ACT)
WAIT FOR S_READY
;ENDFOLD

;FOLD ; SWP_60_5110;%{PE}%R2.2,%MKUKATPBASIS,%CCOMMENT,%VNORMAL,%P 2: SWP_60_5110
;ENDFOLD
;FOLD PTP swp_60_5110 PDAT58 SPOT Gun= 1 RETR CLS PgNo1= 101 ACTIVE= 1 Tool[1]:GUN C1 Base[1]:Actros ;%{PE}%R 4.1.12,%MKUKATPSPOT,%CSPOT,%VPTP,%P 1:PTP, 2:swp_60_5110, 3:, 5:100, 7:PDAT58, 10:1, 12:#FIRST, 14:#CLO, 16:101, 18:1, 20:0, 22:0, 24:1, 25:NORMAL
$BWDSTART = FALSE
PDAT_ACT=PPDAT58
BAS(#PTP_DAT)
FDAT_ACT=Fswp_60_5110
BAS(#FRAMES)
BAS(#VEL_PTP,PPDAT58.VEL)
S_ACT.GUN=1
S_ACT.PAIR=SDEFAULT.PAIR
S_ACT.RETR=#CLO
S_ACT.CLO_TM=1
S_ACT.PGNO1=101
S_ACT.PGNO2=SDEFAULT.PGNO2
S_ACT.PRESS1=SDEFAULT.PRESS1
S_ACT.PRESS2=SDEFAULT.PRESS2
S_READY=FALSE
PTP Xswp_60_5110
USERSPOT(#SPOT, S_ACT)
WAIT FOR S_READY
;ENDFOLD

;FOLD ; SWP_60_5112;%{PE}%R2.2,%MKUKATPBASIS,%CCOMMENT,%VNORMAL,%P 2: SWP_60_5112
;ENDFOLD
;FOLD PTP swp_60_5112 PDAT59 SPOT Gun= 1 RETR CLS PgNo1= 102 ACTIVE= 1 Tool[1]:GUN C1 Base[1]:Actros ;%{PE}%R 4.1.12,%MKUKATPSPOT,%CSPOT,%VPTP,%P 1:PTP, 2:swp_60_5112, 3:, 5:100, 7:PDAT59, 10:1, 12:#FIRST, 14:#CLO, 16:102, 18:1, 20:0, 22:0, 24:1, 25:NORMAL
$BWDSTART = FALSE
PDAT_ACT=PPDAT59
BAS(#PTP_DAT)
FDAT_ACT=Fswp_60_5112
BAS(#FRAMES)
BAS(#VEL_PTP,PPDAT59.VEL)
S_ACT.GUN=1
S_ACT.PAIR=SDEFAULT.PAIR
S_ACT.RETR=#CLO
S_ACT.CLO_TM=1
S_ACT.PGNO1=102
S_ACT.PGNO2=SDEFAULT.PGNO2
S_ACT.PRESS1=SDEFAULT.PRESS1
S_ACT.PRESS2=SDEFAULT.PRESS2
S_READY=FALSE
PTP Xswp_60_5112
USERSPOT(#SPOT, S_ACT)
WAIT FOR S_READY
;ENDFOLD

;FOLD ; SWP_60_5114;%{PE}%R2.2,%MKUKATPBASIS,%CCOMMENT,%VNORMAL,%P 2: SWP_60_5114
;ENDFOLD
;FOLD PTP swp_60_5114 PDAT60 SPOT Gun= 1 RETR CLS PgNo1= 103 ACTIVE= 1 Tool[1]:GUN C1 Base[1]:Actros ;%{PE}%R 4.1.12,%MKUKATPSPOT,%CSPOT,%VPTP,%P 1:PTP, 2:swp_60_5114, 3:, 5:100, 7:PDAT60, 10:1, 12:#FIRST, 14:#CLO, 16:103, 18:1, 20:0, 22:0, 24:1, 25:NORMAL
$BWDSTART = FALSE
PDAT_ACT=PPDAT60
BAS(#PTP_DAT)
FDAT_ACT=Fswp_60_5114
BAS(#FRAMES)
BAS(#VEL_PTP,PPDAT60.VEL)
S_ACT.GUN=1
S_ACT.PAIR=SDEFAULT.PAIR
S_ACT.RETR=#CLO
S_ACT.CLO_TM=1
S_ACT.PGNO1=103
S_ACT.PGNO2=SDEFAULT.PGNO2
S_ACT.PRESS1=SDEFAULT.PRESS1
S_ACT.PRESS2=SDEFAULT.PRESS2
S_READY=FALSE
PTP Xswp_60_5114
USERSPOT(#SPOT, S_ACT)
WAIT FOR S_READY
;ENDFOLD

;FOLD ; SWP_60_5116;%{PE}%R2.2,%MKUKATPBASIS,%CCOMMENT,%VNORMAL,%P 2: SWP_60_5116
;ENDFOLD
;FOLD PTP swp_60_5116 PDAT61 SPOT Gun= 1 RETR CLS PgNo1= 104 ACTIVE= 1 Tool[1]:GUN C1 Base[1]:Actros ;%{PE}%R 4.1.12,%MKUKATPSPOT,%CSPOT,%VPTP,%P 1:PTP, 2:swp_60_5116, 3:, 5:100, 7:PDAT61, 10:1, 12:#FIRST, 14:#CLO, 16:104, 18:1, 20:0, 22:0, 24:1, 25:NORMAL
$BWDSTART = FALSE
PDAT_ACT=PPDAT61
BAS(#PTP_DAT)
FDAT_ACT=Fswp_60_5116
BAS(#FRAMES)
BAS(#VEL_PTP,PPDAT61.VEL)
S_ACT.GUN=1
S_ACT.PAIR=SDEFAULT.PAIR
S_ACT.RETR=#CLO
S_ACT.CLO_TM=1
S_ACT.PGNO1=104
S_ACT.PGNO2=SDEFAULT.PGNO2
S_ACT.PRESS1=SDEFAULT.PRESS1
S_ACT.PRESS2=SDEFAULT.PRESS2
S_READY=FALSE
PTP Xswp_60_5116
USERSPOT(#SPOT, S_ACT)
WAIT FOR S_READY
;ENDFOLD

;FOLD PTP p1118 CONT Vel= 65 % P_OLP92 Tool[1]:GUN C1 Base[1]:Actros ;%{PE}%R 4.1.16,%MKUKATPBASIS,%CMOVE,%VPTP,%P 1:PTP, 2:p1118, 3:C_PTP, 5:65, 7:P_OLP92
$BWDSTART = FALSE
PDAT_ACT=PP_OLP92
BAS(#PTP_DAT)
FDAT_ACT=Fp1118
BAS(#FRAMES)
BAS(#VEL_PTP,65)
PTP Xp1118 C_PTP
;ENDFOLD
;FOLD PTP p1119 CONT Vel= 80 % P_OLP93 Tool[1]:GUN C1 Base[1]:Actros ;%{PE}%R 4.1.16,%MKUKATPBASIS,%CMOVE,%VPTP,%P 1:PTP, 2:p1119, 3:C_PTP, 5:80, 7:P_OLP93
$BWDSTART = FALSE
PDAT_ACT=PP_OLP93
BAS(#PTP_DAT)
FDAT_ACT=Fp1119
BAS(#FRAMES)
BAS(#VEL_PTP,80)
PTP Xp1119 C_PTP
;ENDFOLD

;FOLD PTP HOME  Vel= 100 % DEFAULT;%{PE}%R 4.1.16,%MKUKATPBASIS,%CMOVE,%VPTP,%P 1:PTP, 2:HOME, 3:, 5:100, 7:DEFAULT
$BWDSTART = FALSE
PDAT_ACT=PDEFAULT
BAS(#PTP_DAT)
FDAT_ACT=FHOME
BAS(#FRAMES)
BAS(#VEL_PTP,100)
$H_POS=XHOME
PTP XHOME
;ENDFOLD

;FOLD OUT 839 'R4 Soldando'  State= FALSE ;%{PE}%R 4.1.16,%MKUKATPBASIS,%COUT,%VOUTX,%P 2:839, 3:'R4 Soldando', 5:FALSE, 6:
$OUT[839]=FALSE
;ENDFOLD
;FOLD OUT 848 'Area de Solda'  State= TRUE ;%{PE}%R 4.1.16,%MKUKATPBASIS,%COUT,%VOUTX,%P 2:848, 3:'Area de Solda', 5:TRUE, 6:
$OUT[848]=TRUE
;ENDFOLD

;FOLD ; END INTERLOCK COM R3;%{PE}%R2.2,%MKUKATPBASIS,%CCOMMENT,%VNORMAL,%P 2: END INTERLOCK COM R3
;ENDFOLD

;FOLD Kollision.Ueberwachung_3_Aus ;%{PE}%MKUKATPUSER
COLLSTOP( 3, 2 )
;ENDFOLD

;FOLD PULSE 844 'R4 solda RESPOT concluida'  State= TRUE CONT  Time= 3 sec;%{PE}%R 4.1.16,%MKUKATPBASIS,%COUT,%VPULSE,%P 2:844, 3:'R4 solda RESPOT concluida', 5:TRUE, 6:CONTINUE, 8:3
CONTINUE
PULSE($OUT[844], TRUE,3)
;ENDFOLD

END

--- ps_604ac_c1.dat ---
&ACCESS RVO1
&REL 76
&COMMENT Resp C1 Actros
DEFDAT  PS_604AC_C1
;FOLD EXTERNAL DECLARATIONS;%{PE}%V2.2.2,%MKUKATPBASIS,%CEXT,%VCOMMON,%P
;FOLD BAS EXT;%{PE}%V2.2.2,%MKUKATPBASIS,%CEXT,%VEXT,%P
EXT  BAS (BAS_COMMAND  :IN,REAL  :IN )
DECL INT SUCCESS
;ENDFOLD
;FOLD A10 EXT;%{E}%V2.2.2,%MKUKATPARC,%CEXT,%VEXT,%P
EXT  A10 (A_CMD_T  :IN,A_STRT_T  :IN,A_WELD_T  :IN,A_END_T  :IN,INT  :IN )
;ENDFOLD
;FOLD A20 EXT;%{E}%V2.2.2,%MKUKATPA20,%CEXT,%VEXT,%P
EXT  A20 (INT  :IN,WELD_ST  :IN,WELD_FI  :IN,INT  :IN )
;ENDFOLD
;FOLD GRIPPER EXT;%{E}%V2.2.2,%MKUKATPGRIPPER,%CEXT,%VEXT,%P
EXT  H50 (INT  :IN,INT  :IN,INT  :IN,GRP_TYP  :IN )
;ENDFOLD
;FOLD SPOT EXT;%{E}%V2.2.2,%MKUKATPSPOT,%CEXT,%VEXT,%P
EXT  USERSPOT (S_COMMAND  :IN,SPOT_TYPE  :IN )
;ENDFOLD
;FOLD TOUCHSENSE EXT;%{E}%V2.2.2,%MKUKATPTS,%CEXT,%VEXT,%P
EXT  H70 (INT  :IN,SRCH_TYP_2  :OUT,E6POS  :IN,SRCH_TYP_3  :IN,SRCH_TYP_2  :IN,SRCH_TYP_2  :IN,SRCH_TYP_2  :IN,SRCH_TYP_2  :IN,SRCH_TYP_2  :IN,INT  :IN )
;ENDFOLD
;FOLD USER EXT;%{}%V2.2.2,%MKUKATPUSER,%CEXT,%VEXT,%P
;Make here your modifications
;ENDFOLD
;ENDFOLD

;# ============ START PATH : swp_p13060r4_all_resp_c1 =============
DECL FDAT Fp1028={TOOL_NO 1,BASE_NO 1,IPO_FRAME #BASE}
DECL PDAT PP_OLP2={VEL 100.0,ACC 100.0,APO_DIST 100.0}
DECL E6POS Xp1028={x 80.6620026,y 661.0,z 154.817993,a -90.3581009,b 25.0825996,c 89.7152023,s 2,t 42}
DECL FDAT Fp1029={TOOL_NO 1,BASE_NO 1,IPO_FRAME #BASE}
DECL PDAT PP_OLP3={VEL 100.0,ACC 100.0,APO_DIST 100.0}
DECL E6POS Xp1029={x 153.5,y 659.439026,z 161.518997,a -90.0,b 24.9999008,c 90.0,s 2,t 42}
DECL FDAT Fp1044={TOOL_NO 1,BASE_NO 1,IPO_FRAME #BASE}
DECL PDAT PP_OLP18={VEL 100.0,ACC 100.0,APO_DIST 100.0}
DECL E6POS Xp1044={x 153.501495,y 688.411987,z 140.910599,a 90.0003128,b 80.4786072,c -89.9995422,s 2,t 10,e1 0.0,e2 0.0,e3 0.0,e4 0.0,e5 0.0,e6 0.0}
DECL FDAT Fp1045={TOOL_NO 1,BASE_NO 1,IPO_FRAME #BASE}
DECL PDAT PP_OLP19={VEL 100.0,ACC 100.0,APO_DIST 100.0}
DECL E6POS Xp1045={x 84.7063293,y 690.305786,z 135.633804,a 90.8388367,b 78.7913589,c -88.8695602,s 2,t 10,e1 0.0,e2 0.0,e3 0.0,e4 0.0,e5 0.0,e6 0.0}
DECL FDAT Fp1046={TOOL_NO 1,BASE_NO 1,IPO_FRAME #BASE}
DECL PDAT PP_OLP20={VEL 100.0,ACC 100.0,APO_DIST 100.0}
DECL E6POS Xp1046={x -120.161499,y 377.841888,z 663.636414,a 179.999405,b 80.9414063,c 1.743155,s 2,t 10,e1 0.0,e2 0.0,e3 0.0,e4 0.0,e5 0.0,e6 0.0}
DECL FDAT Fp1047={TOOL_NO 1,BASE_NO 1,IPO_FRAME #BASE}
DECL PDAT PP_OLP21={VEL 100.0,ACC 100.0,APO_DIST 100.0}
DECL E6POS Xp1047={x 104.399803,y 370.90921,z 627.837708,a 179.998398,b 80.9416504,c 1.74246895,s 2,t 10,e1 0.0,e2 0.0,e3 0.0,e4 0.0,e5 0.0,e6 0.0}
DECL FDAT Fp1059={TOOL_NO 1,BASE_NO 1,IPO_FRAME #BASE}
DECL PDAT PP_OLP33={VEL 100.0,ACC 100.0,APO_DIST 100.0}
DECL E6POS Xp1059={x 153.113693,y 938.565491,z 629.284912,a -173.251007,b 88.1828766,c 18.1556797,s 2,t 11,e1 0.0,e2 0.0,e3 0.0,e4 0.0,e5 0.0,e6 0.0}
DECL FDAT Fp1060={TOOL_NO 1,BASE_NO 1,IPO_FRAME #BASE}
DECL PDAT PP_OLP34={VEL 100.0,ACC 100.0,APO_DIST 100.0}
DECL E6POS Xp1060={x 60.7306786,y 869.160522,z -165.050797,a 87.3986511,b -42.5446091,c -88.7094727,s 2,t 42,e1 0.0,e2 0.0,e3 0.0,e4 0.0,e5 0.0,e6 0.0}
DECL FDAT Fp1061={TOOL_NO 1,BASE_NO 1,IPO_FRAME #BASE}
DECL PDAT PP_OLP35={VEL 100.0,ACC 100.0,APO_DIST 100.0}
DECL E6POS Xp1061={x 193.340195,y 864.937012,z -168.289001,a 85.3944702,b -44.9865303,c -87.6166534,s 2,t 43,e1 0.0,e2 0.0,e3 0.0,e4 0.0,e5 0.0,e6 0.0}
DECL FDAT Fp1066={TOOL_NO 1,BASE_NO 1,IPO_FRAME #BASE}
DECL PDAT PP_OLP40={VEL 100.0,ACC 100.0,APO_DIST 100.0}
DECL E6POS Xp1066={x 189.539505,y 825.125671,z -74.1944885,a 90.000618,b -44.9988785,c -90.000351,s 2,t 43,e1 0.0,e2 0.0,e3 0.0,e4 0.0,e5 0.0,e6 0.0}
DECL FDAT Fp1067={TOOL_NO 1,BASE_NO 1,IPO_FRAME #BASE}
DECL PDAT PP_OLP41={VEL 100.0,ACC 100.0,APO_DIST 10.0}
DECL E6POS Xp1067={x 194.101593,y 795.529602,z -103.865402,a 89.9947205,b -45.0005493,c -89.9940796,s 2,t 43,e1 0.0,e2 0.0,e3 0.0,e4 0.0,e5 0.0,e6 0.0}
DECL FDAT Fp1068={TOOL_NO 1,BASE_NO 1,IPO_FRAME #BASE}
DECL PDAT PP_OLP42={VEL 100.0,ACC 100.0,APO_DIST 100.0}
DECL E6POS Xp1068={x 96.6133499,y 714.691528,z -97.3239136,a 86.2758026,b -45.0000381,c -90.0000076,s 2,t 42,e1 0.0,e2 0.0,e3 0.0,e4 0.0,e5 0.0,e6 0.0}
DECL FDAT Fp1069={TOOL_NO 1,BASE_NO 1,IPO_FRAME #BASE}
DECL PDAT PP_OLP43={VEL 100.0,ACC 100.0,APO_DIST 100.0}
DECL E6POS Xp1069={x 103.871101,y 528.69458,z -88.5402679,a 92.9757919,b -15.2220602,c -88.6328735,s 2,t 42,e1 0.0,e2 0.0,e3 0.0,e4 0.0,e5 0.0,e6 0.0}
DECL FDAT Fp1070={TOOL_NO 1,BASE_NO 1,IPO_FRAME #BASE}
DECL PDAT PP_OLP44={VEL 100.0,ACC 100.0,APO_DIST 100.0}
DECL E6POS Xp1070={x 171.460602,y 442.797699,z -53.9892082,a 89.9995728,b -14.9981699,c -89.999939,s 2,t 43,e1 0.0,e2 0.0,e3 0.0,e4 0.0,e5 0.0,e6 0.0}
DECL FDAT Fp1080={TOOL_NO 1,BASE_NO 1,IPO_FRAME #BASE}
DECL PDAT PP_OLP54={VEL 100.0,ACC 100.0,APO_DIST 100.0}
DECL E6POS Xp1080={x 154.783905,y 31.2954693,z -74.2182388,a -7.13862801,b -89.8308716,c 7.18047905,s 2,t 42,e1 0.0,e2 0.0,e3 0.0,e4 0.0,e5 0.0,e6 0.0}
DECL FDAT Fp1081={TOOL_NO 1,BASE_NO 1,IPO_FRAME #BASE}
DECL PDAT PP_OLP55={VEL 100.0,ACC 100.0,APO_DIST 100.0}
DECL E6POS Xp1081={x -12.4278498,y 32.2284698,z -73.6468735,a -5.86978483,b -89.8321075,c 5.91501522,s 2,t 42,e1 0.0,e2 0.0,e3 0.0,e4 0.0,e5 0.0,e6 0.0}
DECL FDAT Fp1082={TOOL_NO 1,BASE_NO 1,IPO_FRAME #BASE}
DECL PDAT PP_OLP56={VEL 100.0,ACC 100.0,APO_DIST 100.0}
DECL E6POS Xp1082={x 74.5642319,y 348.989014,z 159.877502,a -103.788101,b 72.7951965,c 76.1421432,s 2,t 10,e1 0.0,e2 0.0,e3 0.0,e4 0.0,e5 0.0,e6 0.0}
DECL FDAT Fp1083={TOOL_NO 1,BASE_NO 1,IPO_FRAME #BASE}
DECL PDAT PP_OLP57={VEL 100.0,ACC 100.0,APO_DIST 100.0}
DECL E6POS Xp1083={x 153.375397,y 348.263794,z 154.2798,a -103.788101,b 72.7952576,c 76.142067,s 2,t 10,e1 0.0,e2 0.0,e3 0.0,e4 0.0,e5 0.0,e6 0.0}
DECL FDAT Fp1088={TOOL_NO 1,BASE_NO 1,IPO_FRAME #BASE}
DECL PDAT PP_OLP62={VEL 100.0,ACC 100.0,APO_DIST 100.0}
DECL E6POS Xp1088={x 161.209503,y 467.690887,z 146.881897,a 89.9998932,b 30.0001602,c -89.9999924,s 2,t 10,e1 0.0,e2 0.0,e3 0.0,e4 0.0,e5 0.0,e6 0.0}
DECL FDAT Fp1095={TOOL_NO 1,BASE_NO 1,IPO_FRAME #BASE}
DECL PDAT PP_OLP69={VEL 100.0,ACC 100.0,APO_DIST 100.0}
DECL E6POS Xp1095={x 52.1147499,y 268.363892,z 373.153687,a 86.7343674,b -24.9995594,c -90.0000763,s 2,t 42,e1 0.0,e2 0.0,e3 0.0,e4 0.0,e5 0.0,e6 0.0}
DECL FDAT Fp1096={TOOL_NO 1,BASE_NO 1,IPO_FRAME #BASE}
DECL PDAT PP_OLP70={VEL 100.0,ACC 100.0,APO_DIST 100.0}
DECL E6POS Xp1096={x 77.1791382,y 33.5449905,z 374.27301,a 84.8506699,b 19.8732491,c -89.7877502,s 2,t 42,e1 0.0,e2 0.0,e3 0.0,e4 0.0,e5 0.0,e6 0.0}
DECL FDAT Fp1097={TOOL_NO 1,BASE_NO 1,IPO_FRAME #BASE}
DECL PDAT PP_OLP71={VEL 100.0,ACC 100.0,APO_DIST 100.0}
DECL E6POS Xp1097={x 187.415802,y 35.7948494,z 388.134613,a 84.8514404,b 19.8751297,c -89.785347,s 2,t 43,e1 0.0,e2 0.0,e3 0.0,e4 0.0,e5 0.0,e6 0.0}
DECL FDAT Fp1101={TOOL_NO 1,BASE_NO 1,IPO_FRAME #BASE}
DECL PDAT PP_OLP75={VEL 100.0,ACC 100.0,APO_DIST 100.0}
DECL E6POS Xp1101={x 168.383408,y 93.4980774,z 365.252502,a 89.999733,b 39.9999504,c -89.999939,s 2,t 10,e1 0.0,e2 0.0,e3 0.0,e4 0.0,e5 0.0,e6 0.0}
DECL FDAT Fp1105={TOOL_NO 1,BASE_NO 1,IPO_FRAME #BASE}
DECL PDAT PP_OLP79={VEL 100.0,ACC 100.0,APO_DIST 100.0}
DECL E6POS Xp1105={x 165.498398,y 91.3753815,z 457.869507,a 89.9998932,b -34.999939,c -90.0000229,s 2,t 42,e1 0.0,e2 0.0,e3 0.0,e4 0.0,e5 0.0,e6 0.0}
DECL FDAT Fp1109={TOOL_NO 1,BASE_NO 1,IPO_FRAME #BASE}
DECL PDAT PP_OLP83={VEL 100.0,ACC 100.0,APO_DIST 100.0}
DECL E6POS Xp1109={x 161.582901,y -31.9300804,z 424.666992,a 97.7593384,b -81.4697266,c -100.220703,s 2,t 42,e1 0.0,e2 0.0,e3 0.0,e4 0.0,e5 0.0,e6 0.0}
DECL FDAT Fp1110={TOOL_NO 1,BASE_NO 1,IPO_FRAME #BASE}
DECL PDAT PP_OLP84={VEL 100.0,ACC 100.0,APO_DIST 100.0}
DECL E6POS Xp1110={x -112.833603,y -34.6520119,z 422.809296,a 87.4717865,b -81.54245,c -101.852097,s 2,t 42,e1 0.0,e2 0.0,e3 0.0,e4 0.0,e5 0.0,e6 0.0}
DECL FDAT Fp1111={TOOL_NO 1,BASE_NO 1,IPO_FRAME #BASE}
DECL PDAT PP_OLP85={VEL 100.0,ACC 100.0,APO_DIST 100.0}
DECL E6POS Xp1111={x -15.6992598,y 100.110703,z 618.896973,a 75.6258316,b 19.2815094,c -80.7250214,s 2,t 42,e1 0.0,e2 0.0,e3 0.0,e4 0.0,e5 0.0,e6 0.0}
DECL FDAT Fp1112={TOOL_NO 1,BASE_NO 1,IPO_FRAME #BASE}
DECL PDAT PP_OLP86={VEL 100.0,ACC 100.0,APO_DIST 100.0}
DECL E6POS Xp1112={x 97.317688,y 115.379402,z 636.49408,a 98.2293701,b 73.9533234,c -73.6352921,s 2,t 10,e1 0.0,e2 0.0,e3 0.0,e4 0.0,e5 0.0,e6 0.0}
DECL FDAT Fp1118={TOOL_NO 1,BASE_NO 1,IPO_FRAME #BASE}
DECL PDAT PP_OLP92={VEL 100.0,ACC 100.0,APO_DIST 100.0}
DECL E6POS Xp1118={x 103.829803,y 264.970703,z 641.382629,a -179.996506,b 80.766571,c 1.27263904,s 2,t 10,e1 0.0,e2 0.0,e3 0.0,e4 0.0,e5 0.0,e6 0.0}
DECL FDAT Fp1119={TOOL_NO 1,BASE_NO 1,IPO_FRAME #BASE}
DECL PDAT PP_OLP93={VEL 100.0,ACC 100.0,APO_DIST 100.0}
DECL E6POS Xp1119={x -73.2950668,y 268.947388,z 670.182617,a 179.999603,b 80.7673721,c 1.26863503,s 2,t 10,e1 0.0,e2 0.0,e3 0.0,e4 0.0,e5 0.0,e6 0.0}
DECL E6POS XP1={x -42.0721207,y 844.178101,z 630.121094,a -171.8647,b 88.1585922,c 17.8996296,s 2,t 10,e1 0.0,e2 0.0,e3 0.0,e4 0.0,e5 0.0,e6 0.0}
DECL BASIS_SUGG_T LAST_BASIS={POINT1[] "SWP_60_5195             ",POINT2[] "SWP_60_5195             ",CP_PARAMS[] "CPDAT0                  ",PTP_PARAMS[] "PDAT89                  ",CONT[] "C_PTP                   ",CP_VEL[] "2.0                     ",PTP_VEL[] "65                      "}
DECL FDAT FP1={TOOL_NO 1,BASE_NO 1,IPO_FRAME #BASE}
DECL PDAT PPDAT1={VEL 100.0,ACC 100.0,APO_DIST 10.0}
DECL PDAT PPDAT2={VEL 60.0,ACC 100.0,APO_DIST 100.0}
DECL PDAT PPDAT3={VEL 60.0,ACC 100.0,APO_DIST 100.0}
DECL PDAT PPDAT4={VEL 60.0,ACC 100.0,APO_DIST 100.0}
DECL PDAT PPDAT5={VEL 60.0,ACC 100.0,APO_DIST 100.0}
DECL PDAT PPDAT6={VEL 60.0,ACC 100.0,APO_DIST 100.0}
DECL PDAT PPDAT7={VEL 60.0,ACC 100.0,APO_DIST 100.0}
DECL PDAT PPDAT8={VEL 60.0,ACC 100.0,APO_DIST 100.0}
DECL PDAT PPDAT9={VEL 60.0,ACC 100.0,APO_DIST 100.0}
DECL PDAT PPDAT10={VEL 60.0,ACC 100.0,APO_DIST 100.0}
DECL PDAT PPDAT11={VEL 60.0,ACC 100.0,APO_DIST 100.0}
DECL PDAT PPDAT12={VEL 60.0,ACC 100.0,APO_DIST 100.0}
DECL PDAT PPDAT13={VEL 60.0,ACC 100.0,APO_DIST 100.0}
DECL PDAT PPDAT14={VEL 60.0,ACC 100.0,APO_DIST 100.0}
DECL PDAT PPDAT15={VEL 60.0,ACC 100.0,APO_DIST 100.0}
DECL PDAT PPDAT16={VEL 60.0,ACC 100.0,APO_DIST 100.0}
DECL PDAT PPDAT17={VEL 60.0,ACC 100.0,APO_DIST 100.0}
DECL PDAT PPDAT18={VEL 60.0,ACC 100.0,APO_DIST 100.0}
DECL PDAT PPDAT19={VEL 60.0,ACC 100.0,APO_DIST 100.0}
DECL PDAT PPDAT20={VEL 60.0,ACC 100.0,APO_DIST 100.0}
DECL PDAT PPDAT21={VEL 60.0,ACC 100.0,APO_DIST 100.0}
DECL PDAT PPDAT22={VEL 60.0,ACC 100.0,APO_DIST 100.0}
DECL PDAT PPDAT23={VEL 60.0,ACC 100.0,APO_DIST 100.0}
DECL PDAT PPDAT24={VEL 60.0,ACC 100.0,APO_DIST 100.0}
DECL PDAT PPDAT25={VEL 60.0,ACC 100.0,APO_DIST 100.0}
DECL PDAT PPDAT26={VEL 60.0,ACC 100.0,APO_DIST 100.0}
DECL PDAT PPDAT27={VEL 60.0,ACC 100.0,APO_DIST 100.0}
DECL PDAT PPDAT28={VEL 60.0,ACC 100.0,APO_DIST 100.0}
DECL PDAT PPDAT29={VEL 60.0,ACC 100.0,APO_DIST 100.0}
DECL PDAT PPDAT30={VEL 60.0,ACC 100.0,APO_DIST 100.0}
DECL PDAT PPDAT31={VEL 60.0,ACC 100.0,APO_DIST 100.0}
DECL PDAT PPDAT33={VEL 60.0,ACC 100.0,APO_DIST 100.0}
DECL PDAT PPDAT34={VEL 60.0,ACC 100.0,APO_DIST 100.0}
DECL PDAT PPDAT35={VEL 60.0,ACC 100.0,APO_DIST 100.0}
DECL PDAT PPDAT36={VEL 60.0,ACC 100.0,APO_DIST 100.0}
DECL PDAT PPDAT37={VEL 60.0,ACC 100.0,APO_DIST 100.0}
DECL PDAT PPDAT38={VEL 60.0,ACC 100.0,APO_DIST 100.0}
DECL PDAT PPDAT39={VEL 60.0,ACC 100.0,APO_DIST 100.0}
DECL PDAT PPDAT40={VEL 60.0,ACC 100.0,APO_DIST 100.0}
DECL PDAT PPDAT41={VEL 60.0,ACC 100.0,APO_DIST 100.0}
DECL PDAT PPDAT42={VEL 50.0,ACC 100.0,APO_DIST 100.0}
DECL PDAT PPDAT43={VEL 50.0,ACC 100.0,APO_DIST 100.0}
DECL PDAT PPDAT44={VEL 50.0,ACC 100.0,APO_DIST 100.0}
DECL PDAT PPDAT45={VEL 50.0,ACC 100.0,APO_DIST 100.0}
DECL PDAT PPDAT46={VEL 50.0,ACC 100.0,APO_DIST 100.0}
DECL PDAT PPDAT47={VEL 50.0,ACC 100.0,APO_DIST 100.0}
DECL PDAT PPDAT48={VEL 50.0,ACC 100.0,APO_DIST 100.0}
DECL PDAT PPDAT49={VEL 50.0,ACC 100.0,APO_DIST 100.0}
DECL PDAT PPDAT50={VEL 50.0,ACC 100.0,APO_DIST 100.0}
DECL PDAT PPDAT51={VEL 50.0,ACC 100.0,APO_DIST 100.0}
DECL PDAT PPDAT52={VEL 50.0,ACC 100.0,APO_DIST 100.0}
DECL PDAT PPDAT53={VEL 50.0,ACC 100.0,APO_DIST 100.0}
DECL PDAT PPDAT54={VEL 50.0,ACC 100.0,APO_DIST 100.0}
DECL PDAT PPDAT55={VEL 50.0,ACC 100.0,APO_DIST 100.0}
DECL PDAT PPDAT56={VEL 50.0,ACC 100.0,APO_DIST 100.0}
DECL PDAT PPDAT57={VEL 50.0,ACC 100.0,APO_DIST 100.0}
DECL PDAT PPDAT58={VEL 50.0,ACC 100.0,APO_DIST 100.0}
DECL PDAT PPDAT59={VEL 50.0,ACC 100.0,APO_DIST 100.0}
DECL PDAT PPDAT60={VEL 50.0,ACC 100.0,APO_DIST 100.0}
DECL PDAT PPDAT61={VEL 50.0,ACC 100.0,APO_DIST 100.0}
DECL E6POS Xswp_60_5070={x 147.576996,y 625.207214,z 147.8564,a -90.0014496,b 25.0073795,c 90.0020599,s 2,t 42,e1 0.0,e2 0.0,e3 0.0,e4 0.0,e5 0.0,e6 0.0}
DECL FDAT Fswp_60_5070={TOOL_NO 1,BASE_NO 1,IPO_FRAME #BASE}
DECL E6POS Xswp_60_5068={x 147.7453,y 624.854675,z 195.222198,a -90.001503,b -0.00187222997,c 89.9983826,s 2,t 42,e1 0.0,e2 0.0,e3 0.0,e4 0.0,e5 0.0,e6 0.0}
DECL FDAT Fswp_60_5068={TOOL_NO 1,BASE_NO 1,IPO_FRAME #BASE}
DECL E6POS Xswp_60_5064={x 146.078903,y 628.714417,z 303.72229,a -90.2994995,b 0.00605009496,c 91.5301514,s 2,t 42,e1 0.0,e2 0.0,e3 0.0,e4 0.0,e5 0.0,e6 0.0}
DECL FDAT Fswp_60_5064={TOOL_NO 1,BASE_NO 1,IPO_FRAME #BASE}
DECL E6POS Xswp_60_5062={x 145.523499,y 629.77887,z 356.739594,a -90.5743027,b -25.8042908,c 90.7785034,s 2,t 42,e1 0.0,e2 0.0,e3 0.0,e4 0.0,e5 0.0,e6 0.0}
DECL FDAT Fswp_60_5062={TOOL_NO 1,BASE_NO 1,IPO_FRAME #BASE}
DECL E6POS Xswp_60_5094={x 144.187393,y 679.255493,z 389.452911,a -122.629402,b -84.4999771,c 121.836304,s 2,t 42,e1 0.0,e2 0.0,e3 0.0,e4 0.0,e5 0.0,e6 0.0}
DECL FDAT Fswp_60_5094={TOOL_NO 1,BASE_NO 1,IPO_FRAME #BASE}
DECL E6POS Xswp_60_5092={x 147.114197,y 792.970886,z 388.260315,a -179.958893,b -87.2228165,c 179.958206,s 2,t 42,e1 0.0,e2 0.0,e3 0.0,e4 0.0,e5 0.0,e6 0.0}
DECL FDAT Fswp_60_5092={TOOL_NO 1,BASE_NO 1,IPO_FRAME #BASE}
DECL E6POS Xswp_60_5090={x 145.0755,y 841.0755,z 387.759491,a -179.994904,b -87.2207108,c 179.993698,s 2,t 42,e1 0.0,e2 0.0,e3 0.0,e4 0.0,e5 0.0,e6 0.0}
DECL FDAT Fswp_60_5090={TOOL_NO 1,BASE_NO 1,IPO_FRAME #BASE}
DECL E6POS Xswp_60_5088={x 146.463898,y 900.921082,z 351.252594,a 90.5984192,b -0.00365373795,c -93.4180222,s 2,t 10,e1 0.0,e2 0.0,e3 0.0,e4 0.0,e5 0.0,e6 0.0}
DECL FDAT Fswp_60_5088={TOOL_NO 1,BASE_NO 1,IPO_FRAME #BASE}
DECL E6POS Xswp_60_5086={x 146.523697,y 899.844482,z 299.625305,a 90.0005569,b -0.000508172088,c -89.9996338,s 2,t 10,e1 0.0,e2 0.0,e3 0.0,e4 0.0,e5 0.0,e6 0.0}
DECL FDAT Fswp_60_5086={TOOL_NO 1,BASE_NO 1,IPO_FRAME #BASE}
DECL E6POS Xswp_60_5082={x 145.656403,y 897.666382,z 191.832596,a 89.9999237,b -0.000562369009,c -89.9995728,s 2,t 10,e1 0.0,e2 0.0,e3 0.0,e4 0.0,e5 0.0,e6 0.0}
DECL FDAT Fswp_60_5082={TOOL_NO 1,BASE_NO 1,IPO_FRAME #BASE}
DECL E6POS Xswp_60_5080={x 146.273102,y 894.982483,z 140.784195,a 90.0142212,b 23.6818695,c -89.985527,s 2,t 10,e1 0.0,e2 0.0,e3 0.0,e4 0.0,e5 0.0,e6 0.0}
DECL FDAT Fswp_60_5080={TOOL_NO 1,BASE_NO 1,IPO_FRAME #BASE}
DECL E6POS Xswp_60_5078={x 148.729996,y 838.536987,z 93.2813263,a 90.0049362,b 72.6683731,c -89.9926682,s 2,t 10,e1 0.0,e2 0.0,e3 0.0,e4 0.0,e5 0.0,e6 0.0}
DECL FDAT Fswp_60_5078={TOOL_NO 1,BASE_NO 1,IPO_FRAME #BASE}
DECL E6POS Xswp_60_5074={x 146.720306,y 730.969788,z 94.5852432,a 89.982193,b 76.1327209,c -90.0116272,s 2,t 10,e1 0.0,e2 0.0,e3 0.0,e4 0.0,e5 0.0,e6 0.0}
DECL FDAT Fswp_60_5074={TOOL_NO 1,BASE_NO 1,IPO_FRAME #BASE}
DECL E6POS Xswp_60_5072={x 146.603302,y 679.73468,z 95.7607498,a 90.0095673,b 79.5479126,c -89.9905777,s 2,t 10,e1 0.0,e2 0.0,e3 0.0,e4 0.0,e5 0.0,e6 0.0}
DECL FDAT Fswp_60_5072={TOOL_NO 1,BASE_NO 1,IPO_FRAME #BASE}
DECL E6POS Xswp_60_5120={x 87.237442,y 373.947906,z 574.174988,a -175.315002,b 87.0737991,c 10.5248804,s 2,t 10,e1 0.0,e2 0.0,e3 0.0,e4 0.0,e5 0.0,e6 0.0}
DECL FDAT Fswp_60_5120={TOOL_NO 1,BASE_NO 1,IPO_FRAME #BASE}
DECL E6POS Xswp_60_5122={x 87.9792328,y 426.627197,z 572.910217,a 176.429199,b 85.4387131,c 1.48755097,s 2,t 10,e1 0.0,e2 0.0,e3 0.0,e4 0.0,e5 0.0,e6 0.0}
DECL FDAT Fswp_60_5122={TOOL_NO 1,BASE_NO 1,IPO_FRAME #BASE}
DECL E6POS Xswp_60_5124={x 90.4681931,y 480.909485,z 571.79718,a 179.696304,b 86.047348,c 4.72831202,s 2,t 10,e1 0.0,e2 0.0,e3 0.0,e4 0.0,e5 0.0,e6 0.0}
DECL FDAT Fswp_60_5124={TOOL_NO 1,BASE_NO 1,IPO_FRAME #BASE}
DECL E6POS Xswp_60_5126={x 93.5677032,y 534.689697,z 571.383728,a 175.629303,b 86.0130692,c 1.12892401,s 2,t 10,e1 0.0,e2 0.0,e3 0.0,e4 0.0,e5 0.0,e6 0.0}
DECL FDAT Fswp_60_5126={TOOL_NO 1,BASE_NO 1,IPO_FRAME #BASE}
DECL E6POS Xswp_60_5128={x 95.3284073,y 589.288086,z 571.44043,a -177.791397,b 87.466568,c 6.43523979,s 2,t 10,e1 0.0,e2 0.0,e3 0.0,e4 0.0,e5 0.0,e6 0.0}
DECL FDAT Fswp_60_5128={TOOL_NO 1,BASE_NO 1,IPO_FRAME #BASE}
DECL E6POS Xswp_60_5130={x 99.9771729,y 647.107178,z 570.551086,a 179.348694,b 87.1756973,c 4.49086714,s 2,t 10,e1 0.0,e2 0.0,e3 0.0,e4 0.0,e5 0.0,e6 0.0}
DECL FDAT Fswp_60_5130={TOOL_NO 1,BASE_NO 1,IPO_FRAME #BASE}
DECL E6POS Xswp_60_5132={x 104.146698,y 698.281799,z 569.89093,a 179.7314,b 86.2630997,c 6.53987694,s 2,t 10,e1 0.0,e2 0.0,e3 0.0,e4 0.0,e5 0.0,e6 0.0}
DECL FDAT Fswp_60_5132={TOOL_NO 1,BASE_NO 1,IPO_FRAME #BASE}
DECL E6POS Xswp_60_5134={x 107.246696,y 753.889404,z 568.630371,a -157.072998,b 89.4791031,c 29.9156704,s 2,t 10,e1 0.0,e2 0.0,e3 0.0,e4 0.0,e5 0.0,e6 0.0}
DECL FDAT Fswp_60_5134={TOOL_NO 1,BASE_NO 1,IPO_FRAME #BASE}
DECL E6POS Xswp_60_5136={x 112.284897,y 804.700989,z 568.130188,a -169.397507,b 88.8463364,c 17.6055794,s 2,t 10,e1 0.0,e2 0.0,e3 0.0,e4 0.0,e5 0.0,e6 0.0}
DECL FDAT Fswp_60_5136={TOOL_NO 1,BASE_NO 1,IPO_FRAME #BASE}
DECL E6POS Xswp_60_5138={x 119.0093,y 855.849487,z 567.74939,a -174.675201,b 87.3247223,c 14.1563501,s 2,t 10,e1 0.0,e2 0.0,e3 0.0,e4 0.0,e5 0.0,e6 0.0}
DECL FDAT Fswp_60_5138={TOOL_NO 1,BASE_NO 1,IPO_FRAME #BASE}
DECL E6POS Xswp_60_5142={x 133.401199,y 942.991577,z 568.208984,a -176.680801,b 87.7705307,c 14.9821901,s 2,t 11,e1 0.0,e2 0.0,e3 0.0,e4 0.0,e5 0.0,e6 0.0}
DECL FDAT Fswp_60_5142={TOOL_NO 1,BASE_NO 1,IPO_FRAME #BASE}
DECL E6POS Xswp_60_5034={x 172.037399,y 868.708374,z -115.175003,a 87.8129807,b -45.1048813,c -89.3794708,s 2,t 43,e1 0.0,e2 0.0,e3 0.0,e4 0.0,e5 0.0,e6 0.0}
DECL FDAT Fswp_60_5034={TOOL_NO 1,BASE_NO 1,IPO_FRAME #BASE}
DECL E6POS Xswp_60_5032={x 171.622101,y 839.368286,z -88.8312836,a 90.0046463,b -44.9968605,c -90.0039673,s 2,t 43,e1 0.0,e2 0.0,e3 0.0,e4 0.0,e5 0.0,e6 0.0}
DECL FDAT Fswp_60_5032={TOOL_NO 1,BASE_NO 1,IPO_FRAME #BASE}
DECL E6POS Xswp_60_5030={x 171.376602,y 812.701782,z -66.5744171,a 90.0020905,b -45.0012207,c -90.0010223,s 2,t 43,e1 0.0,e2 0.0,e3 0.0,e4 0.0,e5 0.0,e6 0.0}
DECL FDAT Fswp_60_5030={TOOL_NO 1,BASE_NO 1,IPO_FRAME #BASE}
DECL E6POS Xswp_60_5024={x 152.167007,y 394.841309,z -3.15799809,a 1.97667301,b -88.8606796,c -0.602044821,s 2,t 42,e1 0.0,e2 0.0,e3 0.0,e4 0.0,e5 0.0,e6 0.0}
DECL FDAT Fswp_60_5024={TOOL_NO 1,BASE_NO 1,IPO_FRAME #BASE}
DECL E6POS Xswp_60_5022={x 151.880798,y 363.505707,z -1.750633,a 0.220150501,b -88.8182907,c 0.126274496,s 2,t 42,e1 0.0,e2 0.0,e3 0.0,e4 0.0,e5 0.0,e6 0.0}
DECL FDAT Fswp_60_5022={TOOL_NO 1,BASE_NO 1,IPO_FRAME #BASE}
DECL E6POS XSWP_60_5018={x 152.003693,y 302.206512,z -1.02023995,a 0.169115707,b -88.7760391,c 0.0428403988,s 2,t 42,e1 0.0,e2 0.0,e3 0.0,e4 0.0,e5 0.0,e6 0.0}
DECL FDAT Fswp_60_5018={TOOL_NO 1,BASE_NO 1,IPO_FRAME #BASE}
DECL PDAT PPDAT65={VEL 60.0,ACC 100.0,APO_DIST 100.0}
DECL E6POS Xswp_60_5012={x 152.031693,y 199.082504,z 0.958868086,a 0.296492904,b -88.7294464,c -0.292802811,s 2,t 42,e1 0.0,e2 0.0,e3 0.0,e4 0.0,e5 0.0,e6 0.0}
DECL FDAT Fswp_60_5012={TOOL_NO 1,BASE_NO 1,IPO_FRAME #BASE}
DECL E6POS Xswp_60_5010={x 151.4702,y 165.086502,z 1.67742705,a 0.0554335006,b -88.1483078,c -0.0410816111,s 2,t 42,e1 0.0,e2 0.0,e3 0.0,e4 0.0,e5 0.0,e6 0.0}
DECL FDAT Fswp_60_5010={TOOL_NO 1,BASE_NO 1,IPO_FRAME #BASE}
DECL E6POS Xswp_60_5008={x 152.475998,y 136.835297,z 1.14260805,a 157.0065,b -89.039978,c -156.951797,s 2,t 42,e1 0.0,e2 0.0,e3 0.0,e4 0.0,e5 0.0,e6 0.0}
DECL FDAT Fswp_60_5008={TOOL_NO 1,BASE_NO 1,IPO_FRAME #BASE}
DECL E6POS Xswp_60_5006={x 150.548203,y 103.8508,z 1.80931699,a 171.778,b -89.1212006,c -171.5811,s 2,t 42,e1 0.0,e2 0.0,e3 0.0,e4 0.0,e5 0.0,e6 0.0}
DECL FDAT Fswp_60_5006={TOOL_NO 1,BASE_NO 1,IPO_FRAME #BASE}
DECL E6POS Xswp_60_5004={x 150.699493,y 67.4835587,z 2.74040103,a 173.974899,b -88.8019867,c -173.899399,s 2,t 42,e1 0.0,e2 0.0,e3 0.0,e4 0.0,e5 0.0,e6 0.0}
DECL FDAT Fswp_60_5004={TOOL_NO 1,BASE_NO 1,IPO_FRAME #BASE}
DECL E6POS Xswp_60_5002={x 151.382996,y 31.2068291,z 3.33408904,a -5.79885387,b -89.8306274,c 5.83878899,s 2,t 42,e1 0.0,e2 0.0,e3 0.0,e4 0.0,e5 0.0,e6 0.0}
DECL FDAT Fswp_60_5002={TOOL_NO 1,BASE_NO 1,IPO_FRAME #BASE}
DECL E6POS Xswp_60_5213={x 151.343506,y 369.240204,z 101.526604,a -0.1158657,b 88.6060333,c 179.870804,s 2,t 10,e1 0.0,e2 0.0,e3 0.0,e4 0.0,e5 0.0,e6 0.0}
DECL FDAT Fswp_60_5213={TOOL_NO 1,BASE_NO 1,IPO_FRAME #BASE}
DECL E6POS Xswp_60_5212={x 151.7733,y 401.47821,z 101.799301,a 42.0237885,b 89.2618637,c -138.023102,s 2,t 10,e1 0.0,e2 0.0,e3 0.0,e4 0.0,e5 0.0,e6 0.0}
DECL FDAT Fswp_60_5212={TOOL_NO 1,BASE_NO 1,IPO_FRAME #BASE}
DECL E6POS Xswp_60_5211={x 151.244995,y 433.247498,z 101.309799,a 91.8052292,b 67.6212311,c -89.2255783,s 2,t 10,e1 0.0,e2 0.0,e3 0.0,e4 0.0,e5 0.0,e6 0.0}
DECL FDAT Fswp_60_5211={TOOL_NO 1,BASE_NO 1,IPO_FRAME #BASE}
DECL E6POS Xswp_60_5210={x 151.626404,y 466.660492,z 112.450104,a 88.7276306,b 44.9445915,c -91.8367233,s 2,t 10,e1 0.0,e2 0.0,e3 0.0,e4 0.0,e5 0.0,e6 0.0}
DECL FDAT Fswp_60_5210={TOOL_NO 1,BASE_NO 1,IPO_FRAME #BASE}
DECL E6POS Xswp_60_5208={x 152.3992,y 496.237,z 169.305298,a 89.2310333,b -0.00395541405,c -91.5945435,s 2,t 10,e1 0.0,e2 0.0,e3 0.0,e4 0.0,e5 0.0,e6 0.0}
DECL FDAT Fswp_60_5208={TOOL_NO 1,BASE_NO 1,IPO_FRAME #BASE}
DECL E6POS Xswp_60_5207={x 150.895401,y 497.958313,z 205.7276,a 89.234169,b -0.00422674417,c -91.6043701,s 2,t 10,e1 0.0,e2 0.0,e3 0.0,e4 0.0,e5 0.0,e6 0.0}
DECL FDAT Fswp_60_5207={TOOL_NO 1,BASE_NO 1,IPO_FRAME #BASE}
DECL E6POS Xswp_60_5201={x 150.152695,y 414.480896,z 407.18631,a -0.953141093,b -89.9668732,c 0.953172028,s 2,t 42,e1 0.0,e2 0.0,e3 0.0,e4 0.0,e5 0.0,e6 0.0}
DECL FDAT Fswp_60_5201={TOOL_NO 1,BASE_NO 1,IPO_FRAME #BASE}
DECL E6POS Xswp_60_5199={x 151.927795,y 378.551788,z 408.322906,a 0.148779497,b -88.8437576,c -0.146708906,s 2,t 42,e1 0.0,e2 0.0,e3 0.0,e4 0.0,e5 0.0,e6 0.0}
DECL FDAT Fswp_60_5199={TOOL_NO 1,BASE_NO 1,IPO_FRAME #BASE}
DECL E6POS Xswp_60_5197={x 151.784195,y 286.854889,z 409.961914,a -88.6835632,b -89.9887695,c 88.6857529,s 2,t 42,e1 0.0,e2 0.0,e3 0.0,e4 0.0,e5 0.0,e6 0.0}
DECL FDAT Fswp_60_5197={TOOL_NO 1,BASE_NO 1,IPO_FRAME #BASE}
DECL E6POS Xswp_60_5225={x 158.397995,y -34.5563507,z 344.27121,a 124.489899,b 89.9991608,c -55.5090294,s 2,t 10,e1 0.0,e2 0.0,e3 0.0,e4 0.0,e5 0.0,e6 0.0}
DECL FDAT Fswp_60_5225={TOOL_NO 1,BASE_NO 1,IPO_FRAME #BASE}
DECL E6POS Xswp_60_5224={x 158.817596,y 21.7541199,z 342.8461,a 7.251441,b 89.9968719,c -172.745102,s 2,t 10,e1 0.0,e2 0.0,e3 0.0,e4 0.0,e5 0.0,e6 0.0}
DECL FDAT Fswp_60_5224={TOOL_NO 1,BASE_NO 1,IPO_FRAME #BASE}
DECL E6POS Xswp_60_5223={x 158.695206,y 78.0512924,z 341.466492,a 90.2649918,b 82.5856476,c -89.9906693,s 2,t 10,e1 0.0,e2 0.0,e3 0.0,e4 0.0,e5 0.0,e6 0.0}
DECL FDAT Fswp_60_5223={TOOL_NO 1,BASE_NO 1,IPO_FRAME #BASE}
DECL E6POS Xswp_60_5222={x 158.139496,y 119.4897,z 377.400085,a 90.8429031,b 1.34442997,c -89.9818115,s 2,t 42,e1 0.0,e2 0.0,e3 0.0,e4 0.0,e5 0.0,e6 0.0}
DECL FDAT Fswp_60_5222={TOOL_NO 1,BASE_NO 1,IPO_FRAME #BASE}
DECL E6POS Xswp_60_5221={x 156.334198,y 122.213203,z 413.713715,a 90.8429565,b 0.313530207,c -89.9971924,s 2,t 42,e1 0.0,e2 0.0,e3 0.0,e4 0.0,e5 0.0,e6 0.0}
DECL FDAT Fswp_60_5221={TOOL_NO 1,BASE_NO 1,IPO_FRAME #BASE}
DECL E6POS Xswp_60_5220={x 156.435806,y 121.998398,z 447.941193,a 89.9984589,b 0.1692321,c -89.999733,s 2,t 42,e1 0.0,e2 0.0,e3 0.0,e4 0.0,e5 0.0,e6 0.0}
DECL FDAT Fswp_60_5220={TOOL_NO 1,BASE_NO 1,IPO_FRAME #BASE}
DECL E6POS Xswp_60_5239={x 156.396103,y 80.2576828,z 480.775696,a -179.545105,b -88.6039429,c 179.559204,s 2,t 42,e1 0.0,e2 0.0,e3 0.0,e4 0.0,e5 0.0,e6 0.0}
DECL FDAT Fswp_60_5239={TOOL_NO 1,BASE_NO 1,IPO_FRAME #BASE}
DECL E6POS Xswp_60_5238={x 156.501099,y 28.8502007,z 482.382996,a -179.742096,b -87.9393082,c 179.761597,s 2,t 42,e1 0.0,e2 0.0,e3 0.0,e4 0.0,e5 0.0,e6 0.0}
DECL FDAT Fswp_60_5238={TOOL_NO 1,BASE_NO 1,IPO_FRAME #BASE}
DECL E6POS Xswp_60_5237={x 156.747101,y -30.8596001,z 482.960999,a -179.471497,b -88.9242172,c 179.4944,s 2,t 42,e1 0.0,e2 0.0,e3 0.0,e4 0.0,e5 0.0,e6 0.0}
DECL FDAT Fswp_60_5237={TOOL_NO 1,BASE_NO 1,IPO_FRAME #BASE}
DECL E6POS Xswp_60_5108={x 80.7516174,y 60.3081398,z 579.792114,a 179.978607,b 86.2582932,c 0.133161694,s 2,t 10,e1 0.0,e2 0.0,e3 0.0,e4 0.0,e5 0.0,e6 0.0}
DECL FDAT Fswp_60_5108={TOOL_NO 1,BASE_NO 1,IPO_FRAME #BASE}
DECL E6POS Xswp_60_5110={x 81.222023,y 115.354301,z 578.918518,a 179.7565,b 86.7256012,c -0.105138302,s 2,t 10,e1 0.0,e2 0.0,e3 0.0,e4 0.0,e5 0.0,e6 0.0}
DECL FDAT Fswp_60_5110={TOOL_NO 1,BASE_NO 1,IPO_FRAME #BASE}
DECL E6POS Xswp_60_5112={x 81.5925064,y 168.955307,z 579.010925,a 176.137894,b 87.4661484,c -5.23424196,s 2,t 10,e1 0.0,e2 0.0,e3 0.0,e4 0.0,e5 0.0,e6 0.0}
DECL FDAT Fswp_60_5112={TOOL_NO 1,BASE_NO 1,IPO_FRAME #BASE}
DECL E6POS Xswp_60_5114={x 82.1743469,y 220.878799,z 577.750671,a 175.380005,b 87.7489929,c -2.05960011,s 2,t 10,e1 0.0,e2 0.0,e3 0.0,e4 0.0,e5 0.0,e6 0.0}
DECL FDAT Fswp_60_5114={TOOL_NO 1,BASE_NO 1,IPO_FRAME #BASE}
DECL E6POS Xswp_60_5116={x 82.4618835,y 273.9841,z 576.812012,a -177.875397,b 87.0930634,c 3.12462592,s 2,t 10,e1 0.0,e2 0.0,e3 0.0,e4 0.0,e5 0.0,e6 0.0}
DECL FDAT Fswp_60_5116={TOOL_NO 1,BASE_NO 1,IPO_FRAME #BASE}
DECL E6POS XP456={x 151.055893,y 873.993286,z 375.974396,a 92.1770935,b -59.0697784,c -92.2716827,s 2,t 42,e1 0.0,e2 0.0,e3 0.0,e4 0.0,e5 0.0,e6 0.0}
DECL FDAT FP456={TOOL_NO 1,BASE_NO 1,IPO_FRAME #BASE}
DECL PDAT PPDAT66={VEL 100.0,ACC 100.0,APO_DIST 100.0}
DECL E6POS XP457={x 184.557404,y 875.905579,z -119.014702,a 85.3778305,b -45.0793114,c -87.6031113,s 2,t 43,e1 0.0,e2 0.0,e3 0.0,e4 0.0,e5 0.0,e6 0.0}
DECL FDAT FP457={TOOL_NO 1,BASE_NO 1,IPO_FRAME #BASE}
DECL PDAT PPDAT67={VEL 100.0,ACC 100.0,APO_DIST 100.0}
DECL E6POS XP463={x 111.082603,y 561.817383,z 586.249695,a -172.985504,b 88.1748962,c 11.2522697,s 2,t 10,e1 0.0,e2 0.0,e3 0.0,e4 0.0,e5 0.0,e6 0.0}
DECL FDAT FP463={TOOL_NO 1,BASE_NO 1,IPO_FRAME #BASE}
DECL PDAT PPDAT72={VEL 100.0,ACC 100.0,APO_DIST 5.0}
DECL E6POS XP465={x 112.942101,y 673.657898,z 575.536499,a -179.998703,b 86.3741226,c 6.37208986,s 2,t 10,e1 0.0,e2 0.0,e3 0.0,e4 0.0,e5 0.0,e6 0.0}
DECL FDAT FP465={TOOL_NO 1,BASE_NO 1,IPO_FRAME #BASE}
DECL PDAT PPDAT74={VEL 100.0,ACC 100.0,APO_DIST 5.0}
DECL E6POS XP466={x 117.7733,y 726.584473,z 574.164612,a -172.903595,b 88.1740723,c 14.1157303,s 2,t 10,e1 0.0,e2 0.0,e3 0.0,e4 0.0,e5 0.0,e6 0.0}
DECL FDAT FP466={TOOL_NO 1,BASE_NO 1,IPO_FRAME #BASE}
DECL PDAT PPDAT75={VEL 100.0,ACC 100.0,APO_DIST 5.0}
DECL E6POS XP467={x 140.145905,y 901.200989,z 574.929321,a -173.270599,b 88.1826019,c 18.1370392,s 2,t 11,e1 0.0,e2 0.0,e3 0.0,e4 0.0,e5 0.0,e6 0.0}
DECL FDAT FP467={TOOL_NO 1,BASE_NO 1,IPO_FRAME #BASE}
DECL PDAT PPDAT76={VEL 100.0,ACC 100.0,APO_DIST 5.0}
DECL E6POS XSWP_60_5206={x 151.252502,y 496.018005,z 243.910904,a 89.607193,b 7.64656782,c -91.7428894,s 2,t 10,e1 0.0,e2 0.0,e3 0.0,e4 0.0,e5 0.0,e6 0.0}
DECL FDAT FSWP_60_5206={TOOL_NO 1,BASE_NO 1,IPO_FRAME #BASE}
DECL PDAT PPDAT78={VEL 60.0,ACC 100.0,APO_DIST 100.0}
DECL E6POS XSWP_60_5205={x 150.698593,y 497.202911,z 288.503387,a 89.9870071,b 4.46940899,c -91.5525131,s 2,t 10,e1 0.0,e2 0.0,e3 0.0,e4 0.0,e5 0.0,e6 0.0}
DECL FDAT FSWP_60_5205={TOOL_NO 1,BASE_NO 1,IPO_FRAME #BASE}
DECL PDAT PPDAT79={VEL 60.0,ACC 100.0,APO_DIST 100.0}
DECL E6POS XSWP_60_5204={x 150.735901,y 495.42981,z 342.286896,a 90.8882294,b 4.29249287,c -91.4886398,s 2,t 42,e1 0.0,e2 0.0,e3 0.0,e4 0.0,e5 0.0,e6 0.0}
DECL FDAT FSWP_60_5204={TOOL_NO 1,BASE_NO 1,IPO_FRAME #BASE}
DECL PDAT PPDAT80={VEL 60.0,ACC 100.0,APO_DIST 100.0}
DECL E6POS XSWP_60_5202={x 148.287201,y 474.969391,z 398.329895,a 90.8485031,b -69.620491,c -91.0470734,s 2,t 42,e1 0.0,e2 0.0,e3 0.0,e4 0.0,e5 0.0,e6 0.0}
DECL FDAT FSWP_60_5202={TOOL_NO 1,BASE_NO 1,IPO_FRAME #BASE}
DECL PDAT PPDAT81={VEL 60.0,ACC 100.0,APO_DIST 100.0}
DECL E6POS XSWP_60_5200={x 148.848099,y 447.841705,z 408.515686,a 91.1680222,b -76.8122635,c -91.2813034,s 2,t 42,e1 0.0,e2 0.0,e3 0.0,e4 0.0,e5 0.0,e6 0.0}
DECL FDAT FSWP_60_5200={TOOL_NO 1,BASE_NO 1,IPO_FRAME #BASE}
DECL PDAT PPDAT82={VEL 60.0,ACC 100.0,APO_DIST 100.0}
DECL E6POS XSWP_60_5198={x 152.100494,y 344.522186,z 409.03241,a -0.250571609,b -89.2593689,c 0.237192497,s 2,t 42,e1 0.0,e2 0.0,e3 0.0,e4 0.0,e5 0.0,e6 0.0}
DECL FDAT FSWP_60_5198={TOOL_NO 1,BASE_NO 1,IPO_FRAME #BASE}
DECL PDAT PPDAT83={VEL 60.0,ACC 100.0,APO_DIST 100.0}
DECL E6POS XSWP_60_5196={x 150.638702,y 247.124496,z 409.974915,a -178.252594,b -88.0717163,c 177.947006,s 2,t 42,e1 0.0,e2 0.0,e3 0.0,e4 0.0,e5 0.0,e6 0.0}
DECL FDAT FSWP_60_5196={TOOL_NO 1,BASE_NO 1,IPO_FRAME #BASE}
DECL PDAT PPDAT84={VEL 60.0,ACC 100.0,APO_DIST 100.0}
DECL E6POS XSWP_60_5203={x 157.876297,y 227.370605,z 379.019501,a -90.5328522,b -40.9386292,c 90.55439,s 2,t 42,e1 0.0,e2 0.0,e3 0.0,e4 0.0,e5 0.0,e6 0.0}
DECL FDAT FSWP_60_5203={TOOL_NO 1,BASE_NO 1,IPO_FRAME #BASE}
DECL PDAT PPDAT85={VEL 100.0,ACC 100.0,APO_DIST 100.0}
DECL E6POS XSWP_60_5194={x 152.579498,y 200.8992,z 363.247711,a -90.3686371,b -29.1460094,c 90.4061737,s 2,t 42,e1 0.0,e2 0.0,e3 0.0,e4 0.0,e5 0.0,e6 0.0}
DECL FDAT FSWP_60_5194={TOOL_NO 1,BASE_NO 1,IPO_FRAME #BASE}
DECL PDAT PPDAT86={VEL 60.0,ACC 100.0,APO_DIST 100.0}
DECL E6POS XSWP_60_5193={x 150.732605,y 199.847397,z 344.079803,a -90.4965286,b -37.9368401,c 90.530632,s 2,t 42,e1 0.0,e2 0.0,e3 0.0,e4 0.0,e5 0.0,e6 0.0}
DECL FDAT FSWP_60_5193={TOOL_NO 1,BASE_NO 1,IPO_FRAME #BASE}
DECL PDAT PPDAT87={VEL 60.0,ACC 100.0,APO_DIST 100.0}
DECL E6POS XSWP_60_5192={x 152.541107,y 193.543701,z 319.314514,a -90.5317764,b -40.9352493,c 90.5554428,s 2,t 42,e1 0.0,e2 0.0,e3 0.0,e4 0.0,e5 0.0,e6 0.0}
DECL FDAT FSWP_60_5192={TOOL_NO 1,BASE_NO 1,IPO_FRAME #BASE}
DECL PDAT PPDAT88={VEL 60.0,ACC 100.0,APO_DIST 100.0}
DECL E6POS XSWP_60_5195={x 157.894302,y 215.755707,z 262.873108,a -90.5324326,b -40.9363899,c 90.5561905,s 2,t 42,e1 0.0,e2 0.0,e3 0.0,e4 0.0,e5 0.0,e6 0.0}
DECL FDAT FSWP_60_5195={TOOL_NO 1,BASE_NO 1,IPO_FRAME #BASE}
DECL PDAT PPDAT89={VEL 100.0,ACC 100.0,APO_DIST 100.0}
DECL SPOT_SUGG_T LAST_SPOT={GUN[] " 1                      ",RETR_CMD[] "#OPN                    ",CHOISE[] "#FIRST                  ",CLO_TM[] "1                       ",PGNO1[] " 1                      ",PRESS1[] "0                       ",PGNO2[] " 1                      ",PRESS2[] "0                       ",SPOT_PARAMS[] "NORMAL                  "}
ENDDAT
